// TwinCAT 3 PLC project BASF_RecipeCode_PLC
// ProgramVersion: 3.1.4022.4
// libraries:
//   Tc2_ModbusSrv, * (Beckhoff Automation GmbH)
//   Tc2_Standard, * (Beckhoff Automation GmbH)
//   Tc2_System, * (Beckhoff Automation GmbH)
//   Tc2_Utilities, * (Beckhoff Automation GmbH)
//   Tc3_Module, * (Beckhoff Automation GmbH)
// project tree:
//   AlarmUnit/ AlarmHandler.TcPOU, AlarmLogic.TcPOU, AlarmParametersProvider.TcPOU, DisableMaxAndMinAlarms.TcPOU
//   AlarmUnit/Structures/ AlarmParameters.TcDUT
//   DefaultValueCalculator/ GetDefaultValue.TcPOU
//   DUTs/ EachRecipeStep.TcDUT
//   GVL%27S/ Coupler.TcGVL (not stored), R1.TcGVL (not stored)
//   Helpers/ FB_Scaling.TcPOU, ScaledValueCalculator.TcPOU, LampStatusDecider.TcPOU, PossibilittyLogic.TcPOU, RemainingTimeCalculator.TcPOU, ShutDown.TcPOU
//   HuberHandlers/ HC_HUBER_1.TcPOU
//   JumoHelpers/ DataParser.TcPOU, ParameterParsingValue.TcPOU, StringSwapperForJumoRecorder.TcPOU
//   / Maintask.TcTTO, R1_task.TcTTO
//   POUs/ MAIN.TcPOU, PushToStartLogic.TcPOU
//   ReactorManager/AnalogScaling/ FB_AnalogScaling.TcPOU, I_AnalogScaling.TcIO
//   ReactorManager/ FB_Reactor.TcPOU
//   ReactorManager/HeatingCoolingMachineControl/ I_HeatCoolControl.TcIO
//   ReactorManager/Helpers/ Simulator.TcPOU
//   ReactorManager/MotorControl/ FB_MotorControl.TcPOU, I_MotorControl.TcIO
//   ReactorManager/MotorControl/MotorControlSupportModules/ FB_VfdIOControl.TcPOU
//   ReactorManager/RampLogic/ StirrerRampLogic.TcPOU
//   RecipeModules/ RecipeModule_R1.TcPOU, RecipeModule_R2.TcPOU, RecipeModule_R3.TcPOU, RecipeModule_R4.TcPOU, RecipeModule_R5.TcPOU, RecipeModule_R6.TcPOU

CONFIGURATION BASF_RecipeCode_PLC
    RESOURCE PLC ON TwinCAT3
        TASK Maintask(INTERVAL := T#25000us, PRIORITY := 2);
        TASK R1_task(INTERVAL := T#2ms, PRIORITY := 18);
        PROGRAM MAIN WITH Maintask : MAIN;
    END_RESOURCE
END_CONFIGURATION

// ---- AlarmUnit/Structures/AlarmParameters.TcDUT
TYPE AlarmParameters :
STRUCT
	CurrentParameterValue : REAL;
	MaxParameterLimit : REAL;
	MinParameterLimit : REAL;
	MaxLimitAlarm : BOOL;
	MinLimitAlarm : BOOL;
END_STRUCT
END_TYPE

// ---- DUTs/EachRecipeStep.TcDUT
TYPE EachRecipeStep :
STRUCT

   ///Tags for start block
     HeatCoolModeSelection:BOOL:=0; /// 0-is jacket mode/ 1-is process mode
	 HeatCoolDeltaTemp:DINT:=0; 
	 Started:BOOL:=0;
	 StartedTime:STRING:='';
	 Ended:BOOL:=0;
	 EndedTime:STRING:='';

	///Tags for HeatCoolBlock
	HeatCoolEnabled:BOOL:=0;
	HeatCoolStarted:BOOL:=0;
	HeatCoolStartedTime:STRING:='';
	HeatCoolEnded:BOOL:=0;
	HeatCoolEndedTime:STRING:='';
	HeatCoolSetPointExpression:DINT:=0;
	HeatCoolDuration:DINT:=0;
	HeatCoolOperatingMode:BOOL:=0;
	
	///Tags for StirrerBlock
	StirrerEnabled:BOOL:=0;
	StirrerStarted:BOOL:=0;
	StirrerStartedTime:STRING:='';
	StirrerEnded:BOOL:=0;
	StirrerEndedTime:STRING:='';
	StirrerSetPointExpression:DINT:=0;

	///Tags for DoseBlock	
	DosingEnabled:BOOL:=0;
	DosingStarted:BOOL:=0;
	DosingStartedTime:STRING:='';
	DosingEnded:BOOL:=0;
	DosingEndedTime:STRING:='';
    DosingMaxAmount:REAL:=0;
	DosingStopTemp:DINT:=0;
	DosingResumeTemp:DINT:=0;
	DosingRateSetpointExpression:REAL:=0;
	DosingMinRate:DINT:=0;
	DosingMaxRate:DINT:=0;
	DosingSettlingTime:DINT:=0;
	DosingMinPh:DINT:=0;
	DosingMaxPh:DINT:=0;
	DosingOperatingMode:BOOL:=0;
	
	////Tags for Wait tags
	WaitEnabled:BOOL:=0;
	WaitStarted:BOOL:=0;
	WaitStartedTime:STRING:='';
	WaitEndedTime:STRING:='';
	WaitEnded:BOOL:=0;
	WaitDuration:DINT:=0;
	WaitRemainingSeconds : INT;
	WaitRemainingMinutes : INT;
	WaitRemainingTime : STRING;
	
	//Tags for Centrifuge Block
	CentrifugeEnabled : BOOL;
	CentrifugeStarted : BOOL;
	CentrifugeEnded : BOOL;
	CentrifugeSpeedSetPoint : DINT;
	CentrifugeWaitTime : DINT;
	
	//Tags for Valves Block
	ValvesEnabled : BOOL;
	ValvesStarted : BOOL;
	ValvesEnded : BOOL;
	ValveAStatus : BOOL;
	ValveBStatus : BOOL;
	ValveCStatus : BOOL;
	
	//Tags for AOOD Pump Block
	AOODPumpEnabled : BOOL;
	AOODPumpStarted : BOOL;
	AOODPumpEnded : BOOL;
	Pump1Status : BOOL;
	Pump2Status : BOOL;

END_STRUCT
END_TYPE

// ---- ReactorManager/AnalogScaling/I_AnalogScaling.TcIO
INTERFACE I_AnalogScaling

METHOD ActualSpeed : REAL
VAR_INPUT
	nRawSensorValue		: REAL;
	nLowerScaleValue	: REAL;
	nHigherScaleValue	: REAL;
	nOutputLowerLimit	: REAL;
	nOutPutHigherLimit	: REAL;
END_VAR
END_METHOD

METHOD LoadCell : real
VAR_INPUT
	nRawSensorValue		: REAL;
	nLowerScaleValue	: REAL;
	nHigherScaleValue	: REAL;
	nOutputLowerLimit	: REAL;
	nOutPutHigherLimit	: REAL;
END_VAR
END_METHOD

METHOD pH : real
VAR_INPUT
	nRawSensorValue		: REAL;
	nLowerScaleValue	: REAL;
	nHigherScaleValue	: REAL;
	nOutputLowerLimit	: REAL;
	nOutPutHigherLimit	: REAL;
END_VAR
END_METHOD

METHOD Pressure : REAL
VAR_INPUT
	nRawSensorValue		: REAL;
	nLowerScaleValue	: REAL;
	nHigherScaleValue	: REAL;
	nOutputLowerLimit	: REAL;
	nOutPutHigherLimit	: REAL;
END_VAR
END_METHOD

METHOD Temperature : REAL
VAR_INPUT
	nRawSensorValue		: REAL;
	nLowerScaleValue	: REAL;
	nHigherScaleValue	: REAL;
	nOutputLowerLimit	: REAL;
	nOutPutHigherLimit	: REAL;
END_VAR
END_METHOD

END_INTERFACE

// ---- ReactorManager/HeatingCoolingMachineControl/I_HeatCoolControl.TcIO
INTERFACE I_HeatCoolControl

METHOD SetTemperature
VAR_INPUT
	nSetTemperature	: UINT;
END_VAR
END_METHOD

END_INTERFACE

// ---- ReactorManager/MotorControl/I_MotorControl.TcIO
INTERFACE I_MotorControl

METHOD GetActualSpeed : INT
END_METHOD

PROPERTY RemoteLocalStatus : bool
GET
END_GET
END_PROPERTY

METHOD SetSpeed : BOOL
VAR_INPUT
	nSetSpeed: INT;
END_VAR
END_METHOD

METHOD StartMotor : BOOL
VAR_INPUT
	bStart: BOOL;
END_VAR
END_METHOD

METHOD StopMotor : BOOL
VAR_INPUT
	bStop: BOOL;
END_VAR
END_METHOD

END_INTERFACE

// ---- POUs/MAIN.TcPOU
PROGRAM MAIN
VAR	 
	couplerConnectionStatus			: BOOL := TRUE;
	NullRecipeStepArray 			: ARRAY[0..100] OF EachRecipeStep;
	
	fglocal							: FB_LocalSystemTime;
	System_Time						: TIMESTRUCT;
	currentHour						: STRING;
	currentMinute					: STRING;
	concatenatedHourMinuteString	: STRING;
	scaledValueCalculator			: ScaledValueCalculator;
	ClearRecipeTrig_R1				: R_Trig;	
	
	fbAnalogScaling					: FB_AnalogScaling;
	ipAnalogScaling					: I_AnalogScaling	:= fbAnalogScaling;
	
	fbMotorControl					: FB_MotorControl;
	ipMotorControl					: I_MotorControl := fbMotorControl ;
	
	fbReactor						: FB_Reactor(ipAnalogScaling := ipAnalogScaling,ipMotorControl:= ipMotorControl);
END_VAR

VAR_INPUT
	ReactorEmergencyStatus AT %I* 	: ARRAY[1..6] OF BOOL;
END_VAR



// CALL THE REACTOR INSTANCE
fbReactor();



//Update Coupler Connection Status
IF	Coupler.CouplerConnectionState = 8 THEN
	Coupler.couplerConnectionStatus := TRUE;
ELSE
	Coupler.couplerConnectionStatus := FALSE; 
END_IF

//Code For Reading Current System Date and Time
fglocal(
	sNetID:='',
	bEnable:=TRUE,
	dwCycle:=5,
	dwOpt:=1,
	tTimeOut:=DEFAULT_ADS_TIMEOUT,
	bValid=> ,
	systemTime=>System_Time ,
	tzID=> );
	
//update current hour and minute strings	
currentHour := WORD_TO_STRING(fglocal.systemTime.wHour);
currentMinute := WORD_TO_STRING(fglocal.systemTime.wMinute);
concatenatedHourMinuteString := CONCAT(STR1:=currentHour, STR2:= ':');
concatenatedHourMinuteString := CONCAT(STR1:=concatenatedHourMinuteString, STR2:= currentMinute);

(* Update Used Now Status of Reactors and Other Equipment *)
IF R1.HeatCoolStatusFeedback OR R1.StirrerStatusFeedback THEN
	R1.UsedNow := TRUE;
ELSE	
	R1.UsedNow := FALSE;
END_IF

///CALL RECIPE MODULE-R1
IF R1.RecipeStatus THEN
	RecipeModule_R1();
END_IF
  
////End condition to wipe of the data in structure
	ClearRecipeTrig_R1(clk:=R1.ClearRecipe,q=>);
 IF ClearRecipeTrig_R1.Q  THEN
	R1.RecipeStatus:=FALSE;
	R1.RecipeStep := NullRecipeStepArray;
	R1.ClearRecipe:=FALSE;
	R1.RecipeEnded:=FALSE;
	R1.R1STEPS:=0;
	RecipeModule_R1.DosingTotalizerVolume:=0;
END_IF
   
//Stirre ramp
StirrerRampLogic();

END_PROGRAM

// ---- Helpers/ScaledValueCalculator.TcPOU
FUNCTION_BLOCK ScaledValueCalculator
VAR_INPUT
	nRawInputValue			: INT;
	nInputLowerLimit		: REAL;
	nInputHigherLimit		: REAL;
	nOutputLowerLimit		: REAL;
	nOutputHigherLimit		: REAL;
END_VAR
VAR_OUTPUT
		nScaledValueF		: REAL;
	    nScaledValueD		: INT;
END_VAR
VAR
	 nGain		: REAL;
END_VAR

// Scaling Calculations //

	IF	nRawInputValue	<	0	THEN
		nRawInputValue	:=	0;
	END_IF


	IF	 ((nInputHigherLimit - nInputLowerLimit)	<= 0)	OR
		 ((nOutputHigherLimit  - nOutputLowerLimit)	<= 0)	THEN
		nGain	:=	0;
	ELSE
		nGain:=(((nRawInputValue - nInputLowerLimit) / (nInputHigherLimit - nInputLowerLimit)) * (nOutputHigherLimit  - nOutputLowerLimit)) + nOutputLowerLimit;
	END_IF


		nScaledValueF	:=	nGain;
		nScaledValueD	:=	REAL_TO_INT(nGain);

END_FUNCTION_BLOCK

// ---- ReactorManager/AnalogScaling/FB_AnalogScaling.TcPOU
FUNCTION_BLOCK FB_AnalogScaling IMPLEMENTS I_AnalogScaling
VAR_INPUT
END_VAR
VAR_OUTPUT
END_VAR
VAR
		fbScaling		: FB_Scaling;
END_VAR

;

METHOD ActualSpeed : REAL
VAR_INPUT
	nRawSensorValue		: REAL;
	nLowerScaleValue	: REAL;
	nHigherScaleValue	: REAL;
	nOutputLowerLimit	: REAL;
	nOutPutHigherLimit	: REAL;
END_VAR
THIS^.fbScaling(
	nRawInputValue		:= nRawSensorValue, 
	nInputLowerLimit	:= nLowerScaleValue , 
	nInputHigherLimit	:= nHigherScaleValue, 
	nOutputLowerLimit	:= nOutputLowerLimit, 
	nOutputHigherLimit	:= nOutPutHigherLimit , 
	nScaledValueF		=> ActualSpeed, 
	nScaledValueD		=> );
END_METHOD

METHOD LoadCell : REAL
VAR_INPUT
	nRawSensorValue		: REAL;
	nLowerScaleValue	: REAL;
	nHigherScaleValue	: REAL;
	nOutputLowerLimit	: REAL;
	nOutPutHigherLimit	: REAL;
END_VAR
THIS^.fbScaling(
	nRawInputValue		:= nRawSensorValue, 
	nInputLowerLimit	:= nLowerScaleValue , 
	nInputHigherLimit	:= nHigherScaleValue, 
	nOutputLowerLimit	:= nOutputLowerLimit, 
	nOutputHigherLimit	:= nOutPutHigherLimit , 
	nScaledValueF		=> LoadCell, 
	nScaledValueD		=> );
END_METHOD

METHOD pH : REAL
VAR_INPUT
	nRawSensorValue		: REAL;
	nLowerScaleValue	: REAL;
	nHigherScaleValue	: REAL;
	nOutputLowerLimit	: REAL;
	nOutPutHigherLimit	: REAL;
END_VAR
THIS^.fbScaling(
	nRawInputValue		:= nRawSensorValue, 
	nInputLowerLimit	:= nLowerScaleValue , 
	nInputHigherLimit	:= nHigherScaleValue, 
	nOutputLowerLimit	:= nOutputLowerLimit, 
	nOutputHigherLimit	:= nOutPutHigherLimit , 
	nScaledValueF		=> pH, 
	nScaledValueD		=> );
END_METHOD

METHOD Pressure : REAL
VAR_INPUT
	nRawSensorValue		: REAL;
	nLowerScaleValue	: REAL;
	nHigherScaleValue	: REAL;
	nOutputLowerLimit	: REAL;
	nOutPutHigherLimit	: REAL;
END_VAR
THIS^.fbScaling(
	nRawInputValue		:= nRawSensorValue, 
	nInputLowerLimit	:= nLowerScaleValue , 
	nInputHigherLimit	:= nHigherScaleValue, 
	nOutputLowerLimit	:= nOutputLowerLimit, 
	nOutputHigherLimit	:= nOutPutHigherLimit , 
	nScaledValueF		=> Pressure, 
	nScaledValueD		=> );
END_METHOD

METHOD Temperature : REAL
VAR_INPUT
	nRawSensorValue		: REAL;
	nLowerScaleValue	: REAL;
	nHigherScaleValue	: REAL;
	nOutputLowerLimit	: REAL;
	nOutPutHigherLimit	: REAL;
END_VAR
THIS^.fbScaling(
	nRawInputValue		:= nRawSensorValue, 
	nInputLowerLimit	:= nLowerScaleValue , 
	nInputHigherLimit	:= nHigherScaleValue, 
	nOutputLowerLimit	:= nOutputLowerLimit, 
	nOutputHigherLimit	:= nOutPutHigherLimit , 
	nScaledValueF		=> Temperature, 
	nScaledValueD		=> );
END_METHOD

END_FUNCTION_BLOCK

// ---- Helpers/FB_Scaling.TcPOU
FUNCTION_BLOCK FB_Scaling
VAR_INPUT
	nRawInputValue: REAL;
	nInputLowerLimit: REAL;
	nInputHigherLimit: REAL;
	nOutputLowerLimit: REAL;
	nOutputHigherLimit: REAL;
END_VAR
VAR_OUTPUT
	nScaledValueF: REAL;
	nScaledValueD: INT;
END_VAR
VAR
	nGain: REAL;
END_VAR

// Scaling Calculations //

	IF	nRawInputValue	<	0	THEN
		nRawInputValue	:=	0;
	END_IF


	IF	 ((nInputHigherLimit - nInputLowerLimit)	<= 0)	OR
		 ((nOutputHigherLimit  - nOutputLowerLimit)	<= 0)	THEN
		nGain	:=	0;
	ELSE
		nGain:=(((nRawInputValue - nInputLowerLimit) / (nInputHigherLimit - nInputLowerLimit)) * (nOutputHigherLimit  - nOutputLowerLimit)) + nOutputLowerLimit;
	END_IF


		nScaledValueF	:=	nGain;
		nScaledValueD	:=	REAL_TO_INT(nGain);

END_FUNCTION_BLOCK

// ---- ReactorManager/MotorControl/FB_MotorControl.TcPOU
FUNCTION_BLOCK FB_MotorControl IMPLEMENTS I_MotorControl
VAR
	fbVfdIOControl: FB_VFDIOControl;
END_VAR

METHOD GetActualSpeed : INT
GetActualSpeed := fbVfdIOControl.nActualSpeed;
END_METHOD

PROPERTY RemoteLocalStatus : BOOL
GET
RemoteLocalStatus := fbVfdIOControl.bRemoteLocalStatus;
END_GET
END_PROPERTY

METHOD SetSpeed : BOOL
VAR_input
	nSetSpeed	: INT;
END_VAR
fbVfdIOControl.nSetSpeed := nSetSpeed;
END_METHOD

METHOD StartMotor : BOOL
VAR_INPUT
	bStart: BOOL;
END_VAR
fbVfdIOControl.bStartMotor := bStart;
END_METHOD

METHOD StopMotor : BOOL
VAR_INPUT
	bStop: BOOL;
END_VAR
fbVfdIOControl.bStopMotor := bStop;
END_METHOD

END_FUNCTION_BLOCK

// ---- ReactorManager/MotorControl/MotorControlSupportModules/FB_VfdIOControl.TcPOU
FUNCTION_BLOCK FB_VfdIOControl
VAR_INPUT
	bStartMotor			AT %Q*: BOOL;
	bStopMotor			AT %Q*: BOOL;
	nSetSpeed 			AT %Q*: INT;
	nActualSpeed		AT %I*: INT;
	bRemoteLocalStatus  AT %I* : BOOL;
END_VAR
VAR_OUTPUT
END_VAR
VAR

END_VAR

END_FUNCTION_BLOCK

// ---- ReactorManager/FB_Reactor.TcPOU
FUNCTION_BLOCK FB_Reactor
VAR_INPUT
	
END_VAR
VAR_OUTPUT
END_VAR
VAR
	simulator : Simulator;
	random_value : REAL;
	timeCounter : INT;
	updateAllParameters : BOOL;
	simulationMode : BOOL;
	
	ipMotorControl		: I_MotorControl;
	ipAnalogScaling		: I_AnalogScaling;
	nMassTemp AT %I*	: INT;
	nVentTemp AT %I*	: INT;
	nVapourTemp	AT %I*	: INT;
	nPressure AT %I*	: INT;
	nReactorpH AT %I*	: INT;
	nScrubberpH AT %I*	: INT;
	nLoadcell AT %I*	: INT;
	nStirrerSpeed AT %I*: INT;
	nLocalTemp			: REAL;
	nLocalTemp1			: REAL;
	nLocalTemp2			: REAL;
	nLocalTemp3 		: REAL;
	nLocalTemp4 		: REAL;
	nLocalTemp5 		: REAL;
	nLocalTemp6 		: REAL;
	nLocalTemp7 		: REAL;	
	nSpeedSetpoint 		: INT;
	nLocalSpeed			: REAL;
	fbScaling			: FB_Scaling;
END_VAR

IF simulationMode THEN
	IF updateAllParameters THEN
		random_value := 0;
		//Update parameters for R1 using Simulator logic
		random_value := 0;
		simulator(CurrentValue := R1.JacketOutletTemperature, TargetValue := DINT_TO_REAL(R1.HeatCoolSetPoint), SimulatedValue => random_value);
		R1.JacketOutletTemperature := REAL_TO_INT(random_value);
		
		simulator(CurrentValue := R1.ReactorMassTemperature, TargetValue := R1.JacketOutletTemperature, SimulatedValue => random_value);
		R1.ReactorMassTemperature := random_value;
		
		random_value := 0;
		simulator(CurrentValue := R1.StirrerCurrentSpeed, TargetValue := DINT_TO_REAL(R1.StirrerSetPoint), SimulatedValue => random_value);
		R1.StirrerCurrentSpeed := REAL_TO_INT(random_value);
		
		//Reset timeCounter
		updateAllParameters := FALSE;
		timeCounter := 0;
	ELSE
		timeCounter := timeCounter + 1;
		IF timeCounter >= 5 THEN
			updateAllParameters := TRUE;
		END_IF
	END_IF
ELSE
	//To Start Motor or Stop Motor
	(*Motor can be controlled from SCADA only if the Remote button is switched on from panel*)
	IF ipMotorControl.RemoteLocalStatus THEN //To check the panel remote status button
		IF R1.StirrerStatus THEN	
			//TO set the speed of the motor
			nLocalSpeed := R1.StirrerSetPoint*70.45;
			nSpeedSetpoint := TO_INT(nLocalSpeed)+6553;
			ipMotorControl.SetSpeed(nSpeedSetpoint);
		ELSE	
			ipMotorControl.SetSpeed(0);
		END_IF
	ELSE
		R1.StirrerStatus := FALSE;
	END_IF
	//========================================================================================================================================================================================================	
	//To call the Huber instance
	HC_HUBER_1();
	
	//Mass Temperature
	nLocalTemp	:= ipAnalogScaling.Temperature(nMassTemp,0,32767,-90,200);
	
	//Vent temp
	nLocalTemp1	:= ipAnalogScaling.Temperature(nVentTemp,0,32767,0,200);
	
	//Vapour temp
	nLocalTemp2	:= ipAnalogScaling.Temperature(nVapourTemp,0,32767,0,200);
	
	//Reactor pressure
	nLocalTemp3	:= ipAnalogScaling.Pressure(nPressure,0,32767,-1,1.5);
	
	//Reactor pH
	nLocalTemp4	:= ipAnalogScaling.pH(nReactorpH,0,32767,0,14);
	
	//Scrubber pH
	nLocalTemp5	:= ipAnalogScaling.pH(nScrubberpH,0,32767,0,14);
	
	//Load cell
	nLocalTemp6	:= ipAnalogScaling.LoadCell(nLoadcell,0,32767,0,150);
	
	//Stirrer actual speed
	nLocalTemp7	:= ipAnalogScaling.ActualSpeed(nLoadcell,0,32767,0,200);
	
		
	R1.ReactorMassTemperature	:= nLocalTemp ;
	R1.VentTemperature			:= nLocalTemp1 ;
	R1.VapourTemperature		:= nLocalTemp2 ;
	R1.Pressure					:= nLocalTemp3 ;
	R1.PHvalue					:= nLocalTemp4 ;
	R1.StirrerCurrentSpeed		:= TO_INT(nLocalTemp7);
	R1.ScrubberpH		:= nLocalTemp5;
	R1.ReactorMass				:= nLocalTemp6;
END_IF

METHOD FB_init : BOOL
VAR_INPUT
	bInitRetains	: BOOL; // if TRUE, the retain variables are initialized (warm start / cold start)
	bInCopyCode		: BOOL;  // if TRUE, the instance afterwards gets moved into the copy code (online change)
	ipMotorControl	: I_MotorControl;
	ipAnalogScaling	: I_AnalogScaling;
END_VAR
IF ipMotorControl <> 0 THEN
	THIS^.ipMotorControl := ipMotorControl;
END_IF

IF ipAnalogScaling <> 0 THEN
	THIS^.ipAnalogScaling := ipAnalogScaling;
END_IF
END_METHOD

END_FUNCTION_BLOCK

// ---- ReactorManager/Helpers/Simulator.TcPOU
FUNCTION_BLOCK Simulator
VAR_INPUT
	CurrentValue : REAL;
	TargetValue : REAL;
END_VAR
VAR_OUTPUT
	SimulatedValue : REAL;
END_VAR
VAR
	random_value : LREAL;
	fb_ran : DRAND;
END_VAR

fb_ran(Seed := 0, Num => random_value);
IF CurrentValue <= TargetValue THEN
	CurrentValue := CurrentValue + LREAL_TO_REAL(STRING_TO_LREAL(LREAL_TO_FMTSTR(random_value, 2, TRUE)));
ELSE
	CurrentValue := CurrentValue - LREAL_TO_REAL(STRING_TO_LREAL(LREAL_TO_FMTSTR(random_value, 2, TRUE)));
END_IF
SimulatedValue := STRING_TO_LREAL(LREAL_TO_FMTSTR(CurrentValue, 2, TRUE)); //Rounding again here to clear any errors above

END_FUNCTION_BLOCK

// ---- HuberHandlers/HC_HUBER_1.TcPOU
PROGRAM HC_HUBER_1
VAR	
	FcHC_2_Write_1	: FB_MBWriteSingleReg;
	FcHC_2_Write_2	: FB_MBWriteSingleReg;
	FcHC_2_Write_3	: FB_MBWriteSingleReg;
	FcHC_2_Write_4	: FB_MBWriteSingleReg;
	FcHC_2_Write_5	: FB_MBWriteSingleReg;
	FcHC_2_Write_6	: FB_MBWriteSingleReg;

	HCComp_2		: WORD;
	HCSelect_2		: WORD;
	HcCirc			: WORD;
	
	HCTempSetpoint_2		: WORD;
	HCReadParameters_2		: ARRAY[0..10] OF INT;

	HuberReadRegs_2			: FB_MBReadRegs;
	HuberReadTimer_2		: TON;
	HuberReadTimer_22		: TON;
	HuberWriteTimer_2		: TON;
	HuberWriteTimer_22		: TON;
END_VAR

//   HUBER_UNISTAT 510_2
//   HC
//   FUNCTION : DATA AQUISITION AND CONTROL
//   
//   COMMUNICATION WITH UNISTAT OVER MODBUS TCP
//   IP : 192.168.0.18


IF R1.HeatCoolStatus THEN 
	HCComp_2:=1;
	HcCirc:=1;
	ELSE
	HCComp_2:=0;
	HcCirc:=0;
END_IF

HCTempSetpoint_2:=DINT_TO_WORD(R1.HeatCoolSetPoint*100);

R1.HeatCoolStatusFeedback:=HCReadParameters_2[10].0;

R1.JacketOutletTemperature:=(INT_TO_REAL(HCReadParameters_2[1])/100);

///Select jacket/process 
IF R1.HeatCoolTemperatureControlType THEN
   HCSelect_2:=1;
   ELSE
   HCSelect_2:=0;	   
   END_IF





HuberReadTimer_2(IN:=NOT HuberReadTimer_22.Q , PT:=T#50MS, Q=> , ET=> );

HuberReadTimer_22(IN:=HuberReadTimer_2.Q , PT:=T#50MS , Q=> , ET=> );



///To read data  from the huber
HuberReadRegs_2(
	sIPAddr:='192.168.0.1' , 
	nTCPPort:=502 , 
	nUnitID:=1 , 
	nQuantity:=11 , 
	nMBAddr:=0 , 
	cbLength:=SIZEOF(HCReadParameters_2) , 
	pDestAddr:=ADR(HCReadParameters_2) , 
	bExecute:=HuberReadTimer_2.Q , 
	tTimeout:=T#5S , 
	bBusy=> , 
	bError=> , 
	nErrId=> , 
	cbRead=> );

HuberWriteTimer_2(IN:=NOT HuberWriteTimer_22.Q  , PT:=T#100MS , Q=> , ET=> );

HuberWriteTimer_22(IN:=HuberWriteTimer_2.Q , PT:=T#100MS, Q=> , ET=> );	
	
	
///To write temperature setpoint to the huber
FcHC_2_Write_1(
	sIPAddr:='192.168.0.1' , 
	nTCPPort:=502 , 
	nUnitID:=1 , 
	nMBAddr:=0 , 
	nValue:=HCTempSetpoint_2 , 
	bExecute:=HuberWriteTimer_2.Q , 
	tTimeout:=T#5S , 
	bBusy=> , 
	bError=> , 
	nErrId=> );	
	
/// jacket/ process selction	
	FcHC_2_Write_2(
	sIPAddr:='192.168.0.1' , 
	nTCPPort:=502 , 
	nUnitID:=1 , 
	nMBAddr:=19 , 
	nValue:=HCSelect_2 , 
	bExecute:=HuberWriteTimer_2.Q , 
	tTimeout:=T#5S , 
	bBusy=> , 
	bError=> , 
	nErrId=> );	
	
		
////To Switch on the machine	
	FcHC_2_Write_4(
	sIPAddr:='192.168.0.1' , 
	nTCPPort:=502 , 
	nUnitID:=1 , 
	nMBAddr:=20 , 
	nValue:=HCComp_2 , 
	bExecute:=HuberWriteTimer_2.Q , 
	tTimeout:=T#5S , 
	bBusy=> , 
	bError=> , 
	nErrId=> );	
	
	
///To switch on the circulation pump		
	FcHC_2_Write_5(
	sIPAddr:='192.168.0.1' , 
	nTCPPort:=502 , 
	nUnitID:=1 , 
	nMBAddr:=21 , 
	nValue:=HcCirc , 
	bExecute:=HuberWriteTimer_2.Q , 
	tTimeout:=T#5S , 
	bBusy=> , 
	bError=> , 
	nErrId=> );	
	
	
	IF 	FcHC_2_Write_5.bExecute OR 	FcHC_2_Write_4.bExecute OR 	FcHC_2_Write_3.bExecute OR 	FcHC_2_Write_2.bExecute OR 	FcHC_2_Write_1.bExecute OR HuberReadRegs_2.bExecute THEN 
///Error daignostics
	  IF HuberreadRegs_2.nErrId <> 0 OR FcHC_2_Write_1.nErrId <> 0 OR  FcHC_2_Write_2.nErrId <> 0 OR
	   FcHC_2_Write_3.nErrId <> 0 OR  FcHC_2_write_4.nErrId <> 0 THEN
	  R1.HeatCoolFailure:=TRUE;
	   ELSE
	  R1.HeatCoolFailure:=FALSE;
	 END_IF
	 END_IF

END_PROGRAM

// ---- RecipeModules/RecipeModule_R1.TcPOU
PROGRAM RecipeModule_R1
VAR
	shutDownFB:Shutdown;
	remainingTimeCalculator : RemainingTimeCalculator;
	
	DosingTick: INT;
	AbortTrig:R_Trig;
END_VAR
VAR_INPUT
	DosingTotalizerVolume: REAL;
END_VAR

IF R1.RecipeStep[0].Started AND R1.RecipeStep[0].StartedTime = '' THEN
	//Update StartedTime
	R1.RecipeStep[0].StartedTime := MAIN.concatenatedHourMinuteString;
END_IF

// Start Block and HC Mode Selection
IF R1.RecipeStep[R1.R1STEPS].Started THEN
  R1.R1STEPS:= R1.R1STEPS+1;
 // R1.AbortRecipe:=FALSE;
  R1.ClearRecipe:=FALSE;
  R1.RecipeEnded:=FALSE;
END_IF  
 
// Check Process or JACKET SELECTION
IF R1.RecipeStep[0].HeatCoolModeSelection THEN
	R1.HeatCoolTemperatureControlType:=TRUE;
	R1.TemperatureControl:=REAL_TO_DINT(R1.ReactorMassTemperature);
ELSE
	R1.HeatCoolTemperatureControlType:=FALSE;	
	R1.TemperatureControl:=REAL_TO_DINT(R1.JacketOutletTemperature);
END_IF

 IF R1.RecipeStep[R1.R1STEPS].HeatcoolEnabled THEN
	R1.HeatCoolSetPoint:=R1.RecipeStep[R1.R1STEPS].HeatCoolSetpointExpression;		
	R1.RecipeStep[R1.R1STEPS].HeatCoolStarted :=TRUE;
	IF R1.RecipeStep[R1.R1STEPS].HeatCoolStartedTime = '' THEN
		R1.RecipeStep[R1.R1STEPS].HeatCoolStartedTime := Main.concatenatedHourMinuteString;
	END_IF
	R1.HeatCoolStatus:=TRUE;
	
		///Check for condition in step  
	 IF ABS(R1.TemperatureControl-R1.RecipeStep[R1.R1STEPS].HeatCoolSetpointExpression )<0.5 THEN
		R1.RecipeStep[R1.R1STEPS].HeatcoolEnded :=TRUE;	
		IF R1.RecipeStep[R1.R1STEPS].HeatCoolEndedTime = '' THEN
			R1.RecipeStep[R1.R1STEPS].HeatCoolEndedTime := Main.concatenatedHourMinuteString;
		END_IF
	 END_IF     	
 END_IF
	
////Recipe block for stirrer
IF R1.RecipeStep[R1.R1STEPS].StirrerEnabled THEN
	R1.StirrerSetPoint:=R1.RecipeStep[R1.R1STEPS].StirrerSetPointExpression;
	R1.StirrerStatus:=TRUE;	
    R1.RecipeStep[R1.R1STEPS].StirrerStarted:=TRUE;
	IF R1.RecipeStep[R1.R1STEPS].StirrerStartedTime = '' THEN
		R1.RecipeStep[R1.R1STEPS].StirrerStartedTime := Main.concatenatedHourMinuteString;
	END_IF
	
	///Check the Actual speed to end the step
      IF ABS(R1.StirrerCurrentSpeed- R1.RecipeStep[R1.R1STEPS].StirrerSetPointExpression)<8 THEN
		R1.RecipeStep[R1.R1STEPS].StirrerEnded:=TRUE;
		IF R1.RecipeStep[R1.R1STEPS].StirrerEndedTime = '' THEN
			R1.RecipeStep[R1.R1STEPS].StirrerEndedTime := Main.concatenatedHourMinuteString;
		END_IF
	  END_IF
	//Check the rpm TO switch off the vfd
	  IF R1.RecipeStep[R1.R1STEPS].StirrerSetPointExpression=0 THEN
		R1.StirrerStatus:=FALSE;	
	  END_IF///
  END_IF 


(*////Wait Block*)
IF R1.RecipeStep[R1.R1STEPS].WaitEnabled AND NOT R1.RecipeStep[R1STEPS].WaitEnded THEN
    R1.RecipeStep[R1.R1STEPS].WaitStarted:=TRUE;
	IF R1.RecipeStep[R1.R1STEPS].WaitStartedTime = '' THEN
		R1.RecipeStep[R1.R1STEPS].WaitStartedTime := Main.concatenatedHourMinuteString;
	END_IF
	R1.WaitTick:=R1.WaitTick+1;
	IF R1.WaitTick=100  THEN
		//Update the Second Tick
		R1.WaitSecondTick:=R1.WaitSecondTick+1;
		R1.WaitTick:=0;
	END_IF
		
	IF  R1.WaitSecondTick=60  THEN
		//Update the Minute Tick
		R1.WaitMinuteTick:=R1.WaitMinuteTick+1;
		R1.WaitSecondTick:=0;
	END_IF	

	//Update the Remaining Time
	remainingTimeCalculator(elapsedSeconds:= R1.WaitSecondTick, elapsedMinutes:= R1.WaitMinuteTick, givenDuration:= DINT_TO_INT(R1.RecipeStep[R1.R1STEPS].WaitDuration), 
							leftOverSeconds=> R1.RecipeStep[R1.R1STEPS].WaitRemainingSeconds, leftOverMinutes=> R1.RecipeStep[R1.R1STEPS].WaitRemainingMinutes);
	R1.RecipeStep[R1.R1STEPS].WaitRemainingTime := INT_TO_STRING(R1.RecipeStep[R1.R1STEPS].WaitRemainingMinutes);
	R1.RecipeStep[R1.R1STEPS].WaitRemainingTime := CONCAT(STR1:= R1.RecipeStep[R1.R1STEPS].WaitRemainingTime, STR2:= ':');
	R1.RecipeStep[R1.R1STEPS].WaitRemainingTime := CONCAT(STR1:= R1.RecipeStep[R1.R1STEPS].WaitRemainingTime, STR2:= INT_TO_STRING(R1.RecipeStep[R1.R1STEPS].WaitRemainingSeconds));
	
	(*///To write ended time*)
	IF ABS(R1.WaitMinuteTick -R1.RecipeStep[R1.R1STEPS].WaitDuration)=0 THEN
		R1.RecipeStep[R1.R1STEPS].WaitEnded:=TRUE;
		IF R1.RecipeStep[R1.R1STEPS].WaitEndedTime = '' THEN
			R1.RecipeStep[R1.R1STEPS].WaitEndedTime := Main.concatenatedHourMinuteString;
		END_IF
		R1.WaitTick:=0;
		R1.WaitSecondTick:=0;
		R1.WaitMinuteTick:=0;
	END_IF
END_IF
	
IF R1.RecipeStep[R1STEPS].DosingEnabled AND NOT R1.RecipeStep[R1STEPS].DosingEnded THEN
	R1.RecipeStep[R1STEPS].DosingStarted := TRUE;
	IF R1.RecipeStep[R1.R1STEPS].DosingStartedTime = '' THEN
		R1.RecipeStep[R1.R1STEPS].DosingStartedTime := Main.concatenatedHourMinuteString;
	END_IF
	//Update Totalized Volume
		IF  R1.DosingPumpStatus_1 THEN
			DosingTick:=DosingTick+1;
		END_IF
		   
	  IF DosingTick=100 THEN
		  DosingTotalizerVolume:=DosingTotalizerVolume+(R1.RecipeStep[R1STEPS].DosingRateSetpointExpression/2.7 * 0.045);	  
	  END_IF
	  
	  IF DosingTick>100 THEN
		  DosingTick:=0;
	  END_IF
	  
	IF DosingTotalizerVolume < R1.RecipeStep[R1STEPS].DosingMaxAmount THEN
		IF R1.DosingPumpStatus_1 THEN
			IF R1.TemperatureControl < R1.RecipeStep[R1STEPS].DosingStopTemp THEN
				R1.DosingPumpStatus_1 := TRUE;
				R1.DosingPumpSetPoint_1 := R1.RecipeStep[R1STEPS].DosingRateSetpointExpression;
			ELSE
				R1.DosingPumpStatus_1 := FALSE;
				R1.DosingPumpSetPoint_1 := 0;
			END_IF
		ELSE
			IF DosingTotalizerVolume = 0 AND R1.TemperatureControl > R1.RecipeStep[R1STEPS].DosingResumeTemp AND R1.TemperatureControl < R1.RecipeStep[R1STEPS].DosingStopTemp THEN
				//Logic for starting Dosing Pump First Time in a Recipe Step
				R1.DosingPumpStatus_1 := TRUE;
				R1.DosingPumpSetPoint_1 := R1.RecipeStep[R1STEPS].DosingRateSetpointExpression;
			END_IF
			
			IF R1.TemperatureControl < R1.RecipeStep[R1STEPS].DosingResumeTemp THEN
				R1.DosingPumpStatus_1 := TRUE;
				R1.DosingPumpSetPoint_1 := R1.RecipeStep[R1STEPS].DosingRateSetpointExpression;
			END_IF
		END_IF
	ELSE
		R1.DosingPumpStatus_1 := FALSE;
		R1.DosingPumpSetPoint_1 := 0;
		R1.RecipeStep[R1STEPS].DosingEnded := TRUE;
		IF R1.RecipeStep[R1.R1STEPS].DosingEndedTime = '' THEN
			R1.RecipeStep[R1.R1STEPS].DosingEndedTime := Main.concatenatedHourMinuteString;
		END_IF
		DosingTick := 0;
		DosingTotalizerVolume:=0;
	END_IF
END_IF

IF R1.R1STEPS>0 THEN 

(*//Step control block To increment to next step*)
 R1.TotalEnabledValue:=BOOL_TO_INT(R1.RecipeStep[R1.R1STEPS].HeatcoolEnabled)+BOOL_TO_INT(R1.RecipeStep[R1.R1STEPS].StirrerEnabled)+BOOL_TO_INT(R1.RecipeStep[R1.R1STEPS].WaitEnabled)+BOOL_TO_INT( R1.RecipeStep[R1.R1STEPS].DosingEnabled);
 R1.TotalEndedValue:=BOOL_TO_INT(R1.RecipeStep[R1.R1STEPS].HeatCoolEnded)+BOOL_TO_INT(R1.RecipeStep[R1.R1STEPS].StirrerEnded)+BOOL_TO_INT(R1.RecipeStep[R1.R1STEPS].WaitEnded)+BOOL_TO_INT( R1.RecipeStep[R1.R1STEPS].DosingEnded);

    IF (R1.TotalEnabledValue - R1.TotalEndedValue)=0 THEN 
		R1.R1STEPS:=R1.R1STEPS+1;
    END_IF
END_IF
  
 (* ///To End the Recipe**)
 IF  R1.NumberOfRecipeSteps = R1.R1STEPS THEN
	 R1.StirrerStatus:=FALSE;
	 R1.StirrerSetPoint:=0;
	 R1.HeatCoolStatus:=FALSE;
	 R1.HeatCoolSetPoint:=0;	
     R1.StepCompleted:=FALSE;	 
	 R1.RecipeEnded:=TRUE;
	 R1.RecipeStatus:=FALSE;
 END_IF
  
(* //TO ABORT RECIPE*)
AbortTrig(CLK:=R1.AbortRecipe,Q=>);
IF AbortTrig.Q THEN
	shutDownFB(GvlIdentifier := 'R1');
	AbortTrig.CLK := FALSE;
END_IF

END_PROGRAM

// ---- Helpers/ShutDown.TcPOU
FUNCTION_BLOCK PUBLIC ShutDown
VAR_INPUT
	GvlIdentifier : STRING;
END_VAR
VAR_OUTPUT
END_VAR
VAR
END_VAR

IF GvlIdentifier = 'R1' THEN
	R1.RecipeStatus		:= FALSE;
	R1.HeatCoolStatus	:= FALSE;
	R1.StirrerStatus	:= FALSE;
	R1.AbortRecipe		:= FALSE;
END_IF;

END_FUNCTION_BLOCK

// ---- Helpers/RemainingTimeCalculator.TcPOU
FUNCTION_BLOCK PUBLIC RemainingTimeCalculator
VAR_INPUT
	elapsedSeconds : INT;
	elapsedMinutes : INT;
	givenDuration : INT; //Assume Duration in Minutes by default
END_VAR
VAR_OUTPUT
	leftOverSeconds : INT;
	leftOverMinutes : INT;
END_VAR
VAR
END_VAR

IF givenDuration <= elapsedMinutes THEN
	leftOverSeconds := 0;
	leftOverMinutes := 0;
ELSE
	leftOverMinutes := givenDuration - elapsedMinutes - 1;
	leftOverSeconds := 60 - elapsedSeconds;
END_IF

END_FUNCTION_BLOCK

// ---- ReactorManager/RampLogic/StirrerRampLogic.TcPOU
PROGRAM StirrerRampLogic

VAR
	i: INT;
	rTime : STRING;
	rMin : DINT;
	rSec : INT;
END_VAR


//// ramp for stirrer R1
IF R1.StirrerStartTimer=1 THEN
	

R1.StirrerTick:=R1.StirrerTick+1;

IF R1.StirrerTick=40  THEN
	R1.StirrerSecondTick:=R1.StirrerSecondTick+1;
	R1.StirrerTick:=0;
END_IF

IF R1.StirrerSecondTick=60  THEN
	R1.StirrerMinuteTick:=R1.StirrerMinuteTick+1;
	R1.StirrerSecondTick:=0;
END_IF

ELSE
	R1.StirrerTick:=0;
	R1.StirrerSecondTick:=0;
	R1.StirrerMinuteTick:=0;
END_IF
// START RAMP

IF R1.StirrerRampStatus THEN
	//initialize ramp parameters if first step
	IF R1.StirrerRampStep = -1 THEN
		R1.StirrerRampStep := R1.StirrerRampStep + 1;
		R1.StirrerRampStarted[R1.StirrerRampStep]:=TRUE;
		R1.StirrerRampStartedTime[R1.StirrerRampStep]:= Main.concatenatedHourMinuteString;
	END_IF
	
	R1.StirrerStatus := TRUE;
	// WRITE RAMP SP TO Stirrer SP	
	R1.StirrerSetPoint:=R1.StirrerRampSetpoint[R1.StirrerRampStep];
	// CHECK IF RPM REACHES SP
	IF ABS(R1.StirrerCurrentSpeed-R1.StirrerRampSetpoint[R1.StirrerRampStep])<5 THEN
		R1.StirrerSPCheck:=1;
		ELSE
		R1.StirrerSPCheck:=0;
	END_IF
	
	R1.StirrerSPCheck_R(CLK:=R1.StirrerSPCheck , Q=>R1.StirrerSPChecktrigger );
	// IF SP REACHED START TIMER
	IF R1.StirrerSPChecktrigger THEN
	R1.StirrerStartTimer:=1;
		
	END_IF
	// CHECK IF HOLD TIME ELAPSED. IF ELAPSED CHECK IF LAST STEP AND END ELSE INCREMENT STEP
	IF (R1.StirrerMinuteTick-R1.StirrerRampTime[R1.StirrerRampStep])=0 THEN
		  R1.StirrerRampEnded[R1.StirrerRampStep]:=1;
		  IF R1.StirrerRampEndedTime[R1.StirrerRampStep] = '' THEN
			 R1.StirrerRampEndedTime[R1.StirrerRampStep]:= Main.concatenatedHourMinuteString;
		  END_IF
		  R1.StirrerRampStep:=R1.StirrerRampStep+1;
		  IF R1.StirrerRampStep=R1.StirrerRampNumberOfSteps THEN
			  R1.StirrerRampStatus:=0;
			  R1.StirrerStartTimer:=0;  
			  ELSE
				R1.StirrerRampStarted[R1.StirrerRampStep]:=1;
				IF R1.StirrerRampStartedTime[R1.StirrerRampStep] = '' THEN
					R1.StirrerRampStartedTime[R1.StirrerRampStep]:= Main.concatenatedHourMinuteString;
				END_IF
				R1.StirrerMinuteTick:=0;
				R1.StirrerStartTimer:=0;  
		  END_IF
	END_IF
	
	//update the remaining time in current step
	rMin := R1.StirrerRampTime[R1.StirrerRampStep] - R1.StirrerMinuteTick - 1;
	IF rMin < 0 THEN
		rMin := 0;
	END_IF
	rSec := 60 - R1.StirrerSecondTick;
	IF rSec = 0 THEN
		rMin := rMin + 1;
	END_IF
	R1.StirrerRampRemainingTime := concat(DINT_TO_STRING(rMin), ':');
	R1.StirrerRampRemainingTime := concat(R1.StirrerRampRemainingTime, DINT_TO_STRING(rSec));
	
	// SKIP OPERATION . IF SKIP PRESSED THEN INCREMENT STEP AFTER CHECKING BOUNDARY CONDN
	R1.StirrerRampSkip(CLK:=R1.StirrerRampStepSkipStatus , Q=>R1.StirrerRampSkipTrigger );
	IF R1.StirrerRampSkipTrigger AND R1.StirrerRampStep<=(R1.StirrerRampNumberOfSteps - 1) THEN
		R1.StirrerRampStepSkipStatus := FALSE; //reset the bit set true by SCADA
		R1.StirrerRampEnded[R1.StirrerRampStep]:=1;
		R1.StirrerRampEndedTime[R1.StirrerRampStep]:= Main.concatenatedHourMinuteString;
		IF R1.StirrerRampStep < R1.StirrerRampNumberOfSteps THEN
			R1.StirrerRampStep:=R1.StirrerRampStep+1;
			R1.StirrerStartTimer:=0;
			R1.StirrerRampStarted[R1.StirrerRampStep]:=1;
			R1.StirrerRampStartedTime[R1.StirrerRampStep]:=Main.concatenatedHourMinuteString;
		ELSE
			// we are in the last step of Ramp. So turn the RampStatus off.
			R1.StirrerRampStatus := FALSE;
		END_IF
	END_IF
	
	// EDIT OPERATION
	R1.StirrerRampEdit(CLK:=R1.StirrerRampStepEditStatus , Q=>R1.StirrerRampEditTrigger );
	IF R1.StirrerRampEditTrigger THEN
		//reset the timer so the step will start again
		R1.StirrerStartTimer:=0;  
	END_IF
	
	R1.StirrerRampClear(clk:= R1.StirrerRampClearStatus, q=>R1.StirrerRampClearStatus);
	IF R1.StirrerRampClearTrigger THEN
		R1.StirrerRampClearStatus := FALSE; //reset the bit set true by SCADA
		R1.StirrerRampStep:=-1;
		R1.StirrerRampStartedTime[i]:='';
		R1.StirrerRampEndedTime[i]:='';
	END_IF
ELSE
	R1.StirrerRampStep:=-1;
	R1.StirrerRampRemainingTime := '';
	FOR i:= 0 TO 7 DO
		R1.StirrerRampStarted[i]:=FALSE;
		R1.StirrerRampEnded[i]:=FALSE;
	END_FOR
END_IF

END_PROGRAM

// ---- AlarmUnit/AlarmHandler.TcPOU
PROGRAM AlarmHandler
VAR
	alarmLogic : AlarmLogic;
	disableAlarms : DisableMaxAndMinAlarms;
END_VAR

IF R1.AlarmsEnabled AND R1.RunningBatchStatus THEN
	alarmLogic(GivenParameterArray := AlarmParametersProvider(CurrentParameterValue := R1.ReactorMassTemperature, MaxParameterLimit := R1.HCTempMaxLimit, MinParameterLimit := R1.HCTempMinLimit),
			   MaxLimitExceeded =>	R1.HCTempMaxLimitExceeded, MinLimitExceeded => R1.HCTempMinLimitExceeded);
		
    alarmLogic(GivenParameterArray := AlarmParametersProvider(CurrentParameterValue := R1.JacketOutletTemperature, MaxParameterLimit := R1.JacketTempMaxLimit, MinParameterLimit := R1.JacketTempMinLimit),
			   MaxLimitExceeded =>	R1.JacketTempMaxLimitExceeded, MinLimitExceeded => R1.jacketTempMinLimitExceeded);	   
ELSE
	(* Disable alarms *)
	disableAlarms(MaxAlarmStatus => R1.HCTempMaxLimitExceeded, MinAlarmStatus => R1.HCTempMinLimitExceeded);
	disableAlarms(MaxAlarmStatus => R1.JacketTempMaxLimitExceeded, MinAlarmStatus => R1.JacketTempMinLimitExceeded);
END_IF


///Reactor-2
IF R2.AlarmsEnabled AND R2.RunningBatchStatus THEN
	alarmLogic(GivenParameterArray := AlarmParametersProvider(CurrentParameterValue := R2.ReactorMassTemperature, MaxParameterLimit := R2.HCTempMaxLimit, MinParameterLimit := R2.HCTempMinLimit),
			   MaxLimitExceeded =>	R2.HCTempMaxLimitExceeded, MinLimitExceeded => R2.HCTempMinLimitExceeded);
			   
    alarmLogic(GivenParameterArray := AlarmParametersProvider(CurrentParameterValue := R2.JacketOutletTemperature, MaxParameterLimit := R2.JacketTempMaxLimit, MinParameterLimit := R2.JacketTempMinLimit),
			   MaxLimitExceeded =>	R2.JacketTempMaxLimitExceeded, MinLimitExceeded => R2.JacketTempMinLimitExceeded);			   
ELSE
	(* Disable alarms *)
	disableAlarms(MaxAlarmStatus => R2.HCTempMaxLimitExceeded, MinAlarmStatus => R2.HCTempMinLimitExceeded);
	disableAlarms(MaxAlarmStatus => R2.JacketTempMaxLimitExceeded, MinAlarmStatus => R2.JacketTempMinLimitExceeded);
END_IF



///Reactor-3
IF R3.AlarmsEnabled AND R3.RunningBatchStatus THEN
	alarmLogic(GivenParameterArray := AlarmParametersProvider(CurrentParameterValue := R3.ReactorMassTemperature, MaxParameterLimit := R3.HCTempMaxLimit, MinParameterLimit := R3.HCTempMinLimit),
			   MaxLimitExceeded =>	R3.HCTempMaxLimitExceeded, MinLimitExceeded => R3.HCTempMinLimitExceeded);
			   
    alarmLogic(GivenParameterArray := AlarmParametersProvider(CurrentParameterValue := R3.JacketOutletTemperature, MaxParameterLimit := R3.JacketTempMaxLimit, MinParameterLimit := R3.JacketTempMinLimit),
			   MaxLimitExceeded =>	R3.JacketTempMaxLimitExceeded, MinLimitExceeded => R3.JacketTempMinLimitExceeded);			   
ELSE
	(* Disable alarms *)
	disableAlarms(MaxAlarmStatus => R3.HCTempMaxLimitExceeded, MinAlarmStatus => R3.HCTempMinLimitExceeded);
	disableAlarms(MaxAlarmStatus => R3.JacketTempMaxLimitExceeded, MinAlarmStatus => R3.JacketTempMinLimitExceeded);
END_IF



///Reactor-4
IF R4.AlarmsEnabled AND R4.RunningBatchStatus THEN
	alarmLogic(GivenParameterArray := AlarmParametersProvider(CurrentParameterValue := R4.ReactorMassTemperature, MaxParameterLimit := R4.HCTempMaxLimit, MinParameterLimit := R4.HCTempMinLimit),
			   MaxLimitExceeded =>	R4.HCTempMaxLimitExceeded, MinLimitExceeded => R4.HCTempMinLimitExceeded);
			   
    alarmLogic(GivenParameterArray := AlarmParametersProvider(CurrentParameterValue := R4.JacketOutletTemperature, MaxParameterLimit := R4.JacketTempMaxLimit, MinParameterLimit := R4.JacketTempMinLimit),
			   MaxLimitExceeded =>	R4.JacketTempMaxLimitExceeded, MinLimitExceeded => R4.JacketTempMinLimitExceeded);			   
ELSE
	(* Disable alarms *)
	disableAlarms(MaxAlarmStatus => R4.HCTempMaxLimitExceeded, MinAlarmStatus => R4.HCTempMinLimitExceeded);
	disableAlarms(MaxAlarmStatus => R4.JacketTempMaxLimitExceeded, MinAlarmStatus => R4.JacketTempMinLimitExceeded);
END_IF




///Reactor-5
IF R5.AlarmsEnabled AND R5.RunningBatchStatus THEN
	alarmLogic(GivenParameterArray := AlarmParametersProvider(CurrentParameterValue := R5.ReactorMassTemperature, MaxParameterLimit := R5.HCTempMaxLimit, MinParameterLimit := R5.HCTempMinLimit),
			   MaxLimitExceeded =>	R5.HCTempMaxLimitExceeded, MinLimitExceeded => R5.HCTempMinLimitExceeded);
			   
    alarmLogic(GivenParameterArray := AlarmParametersProvider(CurrentParameterValue := R5.JacketOutletTemperature, MaxParameterLimit := R5.JacketTempMaxLimit, MinParameterLimit := R5.JacketTempMinLimit),
			   MaxLimitExceeded =>	R5.JacketTempMaxLimitExceeded, MinLimitExceeded => R5.JacketTempMinLimitExceeded);			   
ELSE
	(* Disable alarms *)
	disableAlarms(MaxAlarmStatus => R5.HCTempMaxLimitExceeded, MinAlarmStatus => R5.HCTempMinLimitExceeded);
	disableAlarms(MaxAlarmStatus => R5.JacketTempMaxLimitExceeded, MinAlarmStatus => R5.JacketTempMinLimitExceeded);
END_IF




///Reactor-6
IF R6.AlarmsEnabled AND R6.RunningBatchStatus THEN
	alarmLogic(GivenParameterArray := AlarmParametersProvider(CurrentParameterValue := R6.ReactorMassTemperature, MaxParameterLimit := R6.HCTempMaxLimit, MinParameterLimit := R6.HCTempMinLimit),
			   MaxLimitExceeded =>	R6.HCTempMaxLimitExceeded, MinLimitExceeded => R6.HCTempMinLimitExceeded);
			   
    alarmLogic(GivenParameterArray := AlarmParametersProvider(CurrentParameterValue := R6.JacketOutletTemperature, MaxParameterLimit := R6.JacketTempMaxLimit, MinParameterLimit := R6.JacketTempMinLimit),
			   MaxLimitExceeded =>	R6.JacketTempMaxLimitExceeded, MinLimitExceeded => R6.JacketTempMinLimitExceeded);			   
ELSE
	(* Disable alarms *)
	disableAlarms(MaxAlarmStatus => R6.HCTempMaxLimitExceeded, MinAlarmStatus => R6.HCTempMinLimitExceeded);
	disableAlarms(MaxAlarmStatus => R6.JacketTempMaxLimitExceeded, MinAlarmStatus => R6.JacketTempMinLimitExceeded);
END_IF

END_PROGRAM

// ---- AlarmUnit/AlarmLogic.TcPOU
FUNCTION_BLOCK PUBLIC AlarmLogic
VAR_INPUT
	GivenParameterArray : AlarmParameters;
END_VAR
VAR_OUTPUT
	MaxLimitExceeded : BOOL;
	MinLimitExceeded : BOOL;
END_VAR
VAR
END_VAR

(*
Check if Exceeded bit(Max or Min) was false initially then only write True to Exceeded bit
because overwriting True leads to unnecessary notifications from Plc to Application
*)
IF GivenParameterArray.CurrentParameterValue > GivenParameterArray.MaxParameterLimit AND NOT MaxLimitExceeded THEN
	MaxLimitExceeded := TRUE;
	MinLimitExceeded := FALSE;
ELSIF GivenParameterArray.CurrentParameterValue < GivenParameterArray.MinParameterLimit AND NOT MinLimitExceeded THEN
	MaxLimitExceeded := FALSE;
	MinLimitExceeded := TRUE;
ELSIF GivenParameterArray.CurrentParameterValue <= GivenParameterArray.MaxParameterLimit AND GivenParameterArray.CurrentParameterValue >= GivenParameterArray.MinParameterLimit THEN
	(* Disable the Exceeded bits if current parameter value lies between Max and Min Limits *)
	MaxLimitExceeded := FALSE;
	MinLimitExceeded := FALSE;
END_IF

END_FUNCTION_BLOCK

// ---- AlarmUnit/DisableMaxAndMinAlarms.TcPOU
FUNCTION_BLOCK PUBLIC DisableMaxAndMinAlarms
VAR_INPUT
END_VAR
VAR_OUTPUT
	(* As name suggest force write the Max and Min alarms false *)
	MaxAlarmStatus : BOOL := FALSE;
	MinAlarmStatus : BOOL := FALSE;
END_VAR
VAR
END_VAR

END_FUNCTION_BLOCK

// ---- AlarmUnit/AlarmParametersProvider.TcPOU
FUNCTION AlarmParametersProvider : AlarmParameters
VAR_INPUT
	CurrentParameterValue : REAL;
	MaxParameterLimit : REAL;
	MinParameterLimit : REAL;
END_VAR
VAR
	alarmParameters : AlarmParameters;
END_VAR

alarmParameters.CurrentParameterValue := CurrentParameterValue;
alarmParameters.MaxParameterLimit := MaxParameterLimit;
alarmParameters.MinParameterLimit := MinParameterLimit;

AlarmParametersProvider := alarmParameters;

END_FUNCTION

// ---- DefaultValueCalculator/GetDefaultValue.TcPOU
FUNCTION GetDefaultValue : string
VAR_INPUT
	DataType : STRING;
END_VAR
VAR
	defaultValue : STRING;
END_VAR

IF DataType = 'string' THEN
	defaultValue := '';
END_IF

GetDefaultValue := defaultValue;

END_FUNCTION

// ---- Helpers/LampStatusDecider.TcPOU
FUNCTION_BLOCK PUBLIC LampStatusDecider
VAR_INPUT
	GivenTimer : TON;
	GivenTimer_1: TON;
	Giventimer_2: TON;
	
	CurrentStatus : BOOL;
END_VAR
VAR_OUTPUT
	NewStatus : BOOL;
END_VAR
VAR
END_VAR



	GivenTimer_1(IN:= NOT Giventimer_2.Q,PT:=T#500MS,Q=> );
	
	GivenTimer_2(IN:=GivenTimer_1.Q,PT:=T#500ms,Q=>);
	
	IF GivenTimer_1.Q THEN
	   NewStatus:=TRUE;	
	   ELSE
	   NewStatus:=FALSE;	   
	   END_IF
	
	




//IF GivenTimer.Q THEN
	//NewStatus := NOT CurrentStatus;
//END_IF

END_FUNCTION_BLOCK

// ---- Helpers/PossibilittyLogic.TcPOU
FUNCTION_BLOCK PossibilittyLogic
VAR_INPUT
	TriggerInput:BOOL;
END_VAR
VAR_OUTPUT
	TriggerOutput:BOOL;
END_VAR
VAR
	Counter:INT;
	FalseCounter:int;
	TriggerON:R_TRIG;
	TriggerOFF:F_Trig;
END_VAR


///Increment the counter when the bit is high
TriggerON(CLK:=TriggerInput,q=>);
IF TriggerON.Q THEN
  TriggerOutput:=TRUE;
  FalseCounter:=0;
END_IF
///Decrement the counter when the bit is low
//Increment the countier if the input is continoussly low
IF TriggerInput=FALSE THEN
   FalseCounter:=FalseCounter+1;
   IF  FalseCounter>1000 THEN
	   falseCounter:=0;
   END_IF
END_IF

IF FalseCounter>700 THEN
   TriggerOutput:=FALSE;   
   END_IF

END_FUNCTION_BLOCK

// ---- JumoHelpers/DataParser.TcPOU
FUNCTION_BLOCK PUBLIC DataParser
VAR_INPUT
	GivenArray : ARRAY[0..5] OF REAL;
END_VAR
VAR_OUTPUT
	OutputArray : ARRAY[0..5] OF REAL;
END_VAR
VAR
	i : INT;
END_VAR

FOR i:= 0 TO 5 BY 1 DO
    OutputArray[i] := ParameterParsingValue(GivenArray[i]);
END_FOR;

END_FUNCTION_BLOCK

// ---- JumoHelpers/ParameterParsingValue.TcPOU
FUNCTION ParameterParsingValue : REAL
VAR_INPUT
	InputParameter:REAL;
END_VAR	
VAR
	ParsedStringValue:STRING;
	
END_VAR

//Rounding up the given parameter 
ParsedStringValue:=Lreal_to_fmtstr(InputParameter,1,TRUE);

//Converting  String to real

ParameterParsingValue:=STRING_TO_REAL(ParsedStringValue);

END_FUNCTION

// ---- JumoHelpers/StringSwapperForJumoRecorder.TcPOU
FUNCTION StringSwapperForJumoRecorder : STRING
VAR_INPUT
	GivenString : STRING;
END_VAR
VAR
	i : INT;
	tempString : STRING;
	finalSwappedString : STRING;
	lengthOfGivenString : INT := Len(GivenString);
	tempChar : STRING(255);
END_VAR

IF (lengthOfGivenString MOD 2) <> 0 THEN
	GivenString := concat(GivenString, ' ');
END_IF

FOR i:=1 TO Len(GivenString) BY 2 DO
    IF mid(GivenString, 1, i) = ' ' THEN
		tempString := replace(tempString, ' ', 1, i);
	ELSE
		tempString := replace(tempString, mid(GivenString, 1, i), 1, i);
	END_IF
	
	IF mid(GivenString, 1, i + 1) = ' ' THEN
		tempString := replace(tempString, ' ', 1, i + 1);
	ELSE
		tempString := replace(tempString, mid(GivenString, 1, i + 1), 1, i + 1);
	END_IF
	
	tempChar := mid(tempString, 1, i);
	tempString := replace(tempString, mid(tempString, 1, i + 1), 1, i);
	tempString := replace(tempString, tempChar, 1, i + 1);
	
	finalSwappedString := concat(finalSwappedString, mid(tempString, 1, i));
	finalSwappedString := concat(finalSwappedString, mid(tempString, 1, i + 1));
END_FOR;

StringSwapperForJumoRecorder := finalSwappedString;

END_FUNCTION

// ---- POUs/PushToStartLogic.TcPOU
FUNCTION_BLOCK PushToStartLogic
VAR_INPUT
	StartEquipment:BOOL;
END_VAR
VAR_OUTPUT
	RelayCommandToStart:BOOL;
	RelayCommandToStop:BOOL;
END_VAR
VAR
     StartTrig:R_Trig;
	 Stoptrig:F_Trig;
	
	 StartCounter:INT;
	 StopCounter:INT;	
END_VAR

///Logic for the push button

///Start logic 
StartTrig(CLK:=StartEquipment,q=>);

IF StartTrig.Q THEN
   RelayCommandToStart:=TRUE;
END_IF

IF RelayCommandToStart THEN
   StartCounter:=StartCounter+1;
IF StartCounter=50 THEN
   RelayCommandToSTart:=FALSE;	
   StartCounter:=0;
END_IF
END_IF
   
 ///Stop logic
 StopTrig(CLK:=StartEquipmenT,Q=>);
 IF StopTrig.Q THEN
	RelayCommandToStop:=TRUE;
 END_IF
 
 IF RelayCommandToStop THEN
	StopCounter:=StopCounter+1;
    IF StopCounter=50 THEN
	   RelayCommandToStop:=FALSE;
	   StopCounter:=0;
    END_IF
 END_IF

END_FUNCTION_BLOCK

// ---- RecipeModules/RecipeModule_R2.TcPOU
PROGRAM RecipeModule_R2
VAR
	shutDownFB:Shutdown;
	remainingTimeCalculator : RemainingTimeCalculator;
	
	DosingTick: INT;
	AbortTrig:R_Trig;
END_VAR
VAR_INPUT
	DosingTotalizerVolume: REAL;
END_VAR

IF R2.RecipeStep[0].Started AND R2.RecipeStep[0].StartedTime = '' THEN
	//Update StartedTime
	R2.RecipeStep[0].StartedTime := MAIN.concatenatedHourMinuteString;
END_IF

// Start Block and HC Mode Selection
IF R2.RecipeStep[R2.R2STEPS].Started THEN
  R2.R2STEPS:= R2.R2STEPS+1;
 // R2.AbortRecipe:=FALSE;
  R2.ClearRecipe:=FALSE;
  R2.RecipeEnded:=FALSE;
END_IF  
 
// Check Process or JACKET SELECTION
IF R2.RecipeStep[0].HeatCoolModeSelection THEN
	R2.HeatCoolTemperatureControlType:=TRUE;
	R2.TemperatureControl:=REAL_TO_DINT(R2.ReactorMassTemperature);
ELSE
	R2.HeatCoolTemperatureControlType:=FALSE;	
	R2.TemperatureControl:=REAL_TO_DINT(R2.JacketOutletTemperature);
END_IF

 IF R2.RecipeStep[R2.R2STEPS].HeatcoolEnabled THEN
	R2.HeatCoolSetPoint:=R2.RecipeStep[R2.R2STEPS].HeatCoolSetpointExpression;		
	R2.RecipeStep[R2.R2STEPS].HeatCoolStarted :=TRUE;
	IF R2.RecipeStep[R2.R2STEPS].HeatCoolStartedTime = '' THEN
		R2.RecipeStep[R2.R2STEPS].HeatCoolStartedTime := Main.concatenatedHourMinuteString;
	END_IF
	R2.HeatCoolStatus:=TRUE;
	
		///Check for condition in step  
	 IF ABS(R2.TemperatureControl-R2.RecipeStep[R2.R2STEPS].HeatCoolSetpointExpression )<0.5 THEN
		R2.RecipeStep[R2.R2STEPS].HeatcoolEnded :=TRUE;	
		IF R2.RecipeStep[R2.R2STEPS].HeatCoolEndedTime = '' THEN
			R2.RecipeStep[R2.R2STEPS].HeatCoolEndedTime := Main.concatenatedHourMinuteString;
		END_IF
	 END_IF     	
 END_IF
	
////Recipe block for stirrer
IF R2.RecipeStep[R2.R2STEPS].StirrerEnabled THEN
	R2.StirrerSetPoint:=R2.RecipeStep[R2.R2STEPS].StirrerSetPointExpression;
	R2.StirrerStatus:=TRUE;	
    R2.RecipeStep[R2.R2STEPS].StirrerStarted:=TRUE;
	IF R2.RecipeStep[R2.R2STEPS].StirrerStartedTime = '' THEN
		R2.RecipeStep[R2.R2STEPS].StirrerStartedTime := Main.concatenatedHourMinuteString;
	END_IF
	
	///Check the Actual speed to end the step
      IF ABS(R2.StirrerCurrentSpeed- R2.RecipeStep[R2.R2STEPS].StirrerSetPointExpression)<8 THEN
		R2.RecipeStep[R2.R2STEPS].StirrerEnded:=TRUE;
		IF R2.RecipeStep[R2.R2STEPS].StirrerEndedTime = '' THEN
			R2.RecipeStep[R2.R2STEPS].StirrerEndedTime := Main.concatenatedHourMinuteString;
		END_IF
	  END_IF
	//Check the rpm TO switch off the vfd
	  IF R2.RecipeStep[R2.R2STEPS].StirrerSetPointExpression=0 THEN
		R2.StirrerStatus:=FALSE;	
	  END_IF///
  END_IF 


(*////Wait Block*)
IF R2.RecipeStep[R2.R2STEPS].WaitEnabled AND NOT R2.RecipeStep[R2STEPS].WaitEnded THEN
    R2.RecipeStep[R2.R2STEPS].WaitStarted:=TRUE;
	IF R2.RecipeStep[R2.R2STEPS].WaitStartedTime = '' THEN
		R2.RecipeStep[R2.R2STEPS].WaitStartedTime := Main.concatenatedHourMinuteString;
	END_IF
	R2.WaitTick:=R2.WaitTick+1;
	IF R2.WaitTick=100  THEN
		//Update the Second Tick
		R2.WaitSecondTick:=R2.WaitSecondTick+1;
		R2.WaitTick:=0;
	END_IF
		
	IF  R2.WaitSecondTick=60  THEN
		//Update the Minute Tick
		R2.WaitMinuteTick:=R2.WaitMinuteTick+1;
		R2.WaitSecondTick:=0;
	END_IF	

	//Update the Remaining Time
	remainingTimeCalculator(elapsedSeconds:= R2.WaitSecondTick, elapsedMinutes:= R2.WaitMinuteTick, givenDuration:= DINT_TO_INT(R2.RecipeStep[R2.R2STEPS].WaitDuration), 
							leftOverSeconds=> R2.RecipeStep[R2.R2STEPS].WaitRemainingSeconds, leftOverMinutes=> R2.RecipeStep[R2.R2STEPS].WaitRemainingMinutes);
	R2.RecipeStep[R2.R2STEPS].WaitRemainingTime := INT_TO_STRING(R2.RecipeStep[R2.R2STEPS].WaitRemainingMinutes);
	R2.RecipeStep[R2.R2STEPS].WaitRemainingTime := CONCAT(STR1:= R2.RecipeStep[R2.R2STEPS].WaitRemainingTime, STR2:= ':');
	R2.RecipeStep[R2.R2STEPS].WaitRemainingTime := CONCAT(STR1:= R2.RecipeStep[R2.R2STEPS].WaitRemainingTime, STR2:= INT_TO_STRING(R2.RecipeStep[R2.R2STEPS].WaitRemainingSeconds));
	
	(*///To write ended time*)
	IF ABS(R2.WaitMinuteTick -R2.RecipeStep[R2.R2STEPS].WaitDuration)=0 THEN
		R2.RecipeStep[R2.R2STEPS].WaitEnded:=TRUE;
		IF R2.RecipeStep[R2.R2STEPS].WaitEndedTime = '' THEN
			R2.RecipeStep[R2.R2STEPS].WaitEndedTime := Main.concatenatedHourMinuteString;
		END_IF
		R2.WaitTick:=0;
		R2.WaitSecondTick:=0;
		R2.WaitMinuteTick:=0;
	END_IF
END_IF
	
IF R2.RecipeStep[R2STEPS].DosingEnabled AND NOT R2.RecipeStep[R2STEPS].DosingEnded THEN
	R2.RecipeStep[R2STEPS].DosingStarted := TRUE;
	IF R2.RecipeStep[R2.R2STEPS].DosingStartedTime = '' THEN
		R2.RecipeStep[R2.R2STEPS].DosingStartedTime := Main.concatenatedHourMinuteString;
	END_IF
	//Update Totalized Volume
		IF  R2.DosingPumpStatus_1 THEN
			DosingTick:=DosingTick+1;
		END_IF
		   
	  IF DosingTick=100 THEN
		  DosingTotalizerVolume:=DosingTotalizerVolume+(R2.RecipeStep[R2STEPS].DosingRateSetpointExpression/2.7 * 0.045);	  
	  END_IF
	  
	  IF DosingTick>100 THEN
		  DosingTick:=0;
	  END_IF
	  
	IF DosingTotalizerVolume < R2.RecipeStep[R2STEPS].DosingMaxAmount THEN
		IF R2.DosingPumpStatus_1 THEN
			IF R2.TemperatureControl < R2.RecipeStep[R2STEPS].DosingStopTemp THEN
				R2.DosingPumpStatus_1 := TRUE;
				R2.DosingPumpSetPoint_1 := R2.RecipeStep[R2STEPS].DosingRateSetpointExpression;
			ELSE
				R2.DosingPumpStatus_1 := FALSE;
				R2.DosingPumpSetPoint_1 := 0;
			END_IF
		ELSE
			IF DosingTotalizerVolume = 0 AND R2.TemperatureControl > R2.RecipeStep[R2STEPS].DosingResumeTemp AND R2.TemperatureControl < R2.RecipeStep[R2STEPS].DosingStopTemp THEN
				//Logic for starting Dosing Pump First Time in a Recipe Step
				R2.DosingPumpStatus_1 := TRUE;
				R2.DosingPumpSetPoint_1 := R2.RecipeStep[R2STEPS].DosingRateSetpointExpression;
			END_IF
			
			IF R2.TemperatureControl < R2.RecipeStep[R2STEPS].DosingResumeTemp THEN
				R2.DosingPumpStatus_1 := TRUE;
				R2.DosingPumpSetPoint_1 := R2.RecipeStep[R2STEPS].DosingRateSetpointExpression;
			END_IF
		END_IF
	ELSE
		R2.DosingPumpStatus_1 := FALSE;
		R2.DosingPumpSetPoint_1 := 0;
		R2.RecipeStep[R2STEPS].DosingEnded := TRUE;
		IF R2.RecipeStep[R2.R2STEPS].DosingEndedTime = '' THEN
			R2.RecipeStep[R2.R2STEPS].DosingEndedTime := Main.concatenatedHourMinuteString;
		END_IF
		DosingTick := 0;
		DosingTotalizerVolume:=0;
	END_IF
END_IF

IF R2.R2STEPS>0 THEN 

(*//Step control block To increment to next step*)
 R2.TotalEnabledValue:=BOOL_TO_INT(R2.RecipeStep[R2.R2STEPS].HeatcoolEnabled)+BOOL_TO_INT(R2.RecipeStep[R2.R2STEPS].StirrerEnabled)+BOOL_TO_INT(R2.RecipeStep[R2.R2STEPS].WaitEnabled)+BOOL_TO_INT( R2.RecipeStep[R2.R2STEPS].DosingEnabled);
 R2.TotalEndedValue:=BOOL_TO_INT(R2.RecipeStep[R2.R2STEPS].HeatCoolEnded)+BOOL_TO_INT(R2.RecipeStep[R2.R2STEPS].StirrerEnded)+BOOL_TO_INT(R2.RecipeStep[R2.R2STEPS].WaitEnded)+BOOL_TO_INT( R2.RecipeStep[R2.R2STEPS].DosingEnded);

    IF (R2.TotalEnabledValue - R2.TotalEndedValue)=0 THEN 
		R2.R2STEPS:=R2.R2STEPS+1;
    END_IF
END_IF
  
 (* ///To End the Recipe**)
 IF  R2.NumberOfRecipeSteps = R2.R2STEPS THEN
	 R2.StirrerStatus:=FALSE;
	 R2.StirrerSetPoint:=0;
	 R2.HeatCoolStatus:=FALSE;
	 R2.HeatCoolSetPoint:=0;	
     R2.StepCompleted:=FALSE;	 
	 R2.RecipeEnded:=TRUE;
	 R2.RecipeStatus:=FALSE;
 END_IF
  
(* //TO ABORT RECIPE*)
AbortTrig(CLK:=R2.AbortRecipe,Q=>);
IF AbortTrig.Q THEN
	shutDownFB(GvlIdentifier := 'R2');
	AbortTrig.CLK := FALSE;
END_IF

END_PROGRAM

// ---- RecipeModules/RecipeModule_R3.TcPOU
PROGRAM RecipeModule_R3
VAR
	shutDownFB:Shutdown;
	remainingTimeCalculator : RemainingTimeCalculator;
	
	DosingTick: INT;
	AbortTrig:R_Trig;
END_VAR
VAR_INPUT
	DosingTotalizerVolume: REAL;
END_VAR

IF R3.RecipeStep[0].Started AND R3.RecipeStep[0].StartedTime = '' THEN
	//Update StartedTime
	R3.RecipeStep[0].StartedTime := MAIN.concatenatedHourMinuteString;
END_IF

// Start Block and HC Mode Selection
IF R3.RecipeStep[R3.R3STEPS].Started THEN
  R3.R3STEPS:= R3.R3STEPS+1;
 // R3.AbortRecipe:=FALSE;
  R3.ClearRecipe:=FALSE;
  R3.RecipeEnded:=FALSE;
END_IF  
 
// Check Process or JACKET SELECTION
IF R3.RecipeStep[0].HeatCoolModeSelection THEN
	R3.HeatCoolTemperatureControlType:=TRUE;
	R3.TemperatureControl:=REAL_TO_DINT(R3.ReactorMassTemperature);
ELSE
	R3.HeatCoolTemperatureControlType:=FALSE;	
	R3.TemperatureControl:=REAL_TO_DINT(R3.JacketOutletTemperature);
END_IF

 IF R3.RecipeStep[R3.R3STEPS].HeatcoolEnabled THEN
	R3.HeatCoolSetPoint:=R3.RecipeStep[R3.R3STEPS].HeatCoolSetpointExpression;		
	R3.RecipeStep[R3.R3STEPS].HeatCoolStarted :=TRUE;
	IF R3.RecipeStep[R3.R3STEPS].HeatCoolStartedTime = '' THEN
		R3.RecipeStep[R3.R3STEPS].HeatCoolStartedTime := Main.concatenatedHourMinuteString;
	END_IF
	R3.HeatCoolStatus:=TRUE;
	
		///Check for condition in step  
	 IF ABS(R3.TemperatureControl-R3.RecipeStep[R3.R3STEPS].HeatCoolSetpointExpression )<0.5 THEN
		R3.RecipeStep[R3.R3STEPS].HeatcoolEnded :=TRUE;	
		IF R3.RecipeStep[R3.R3STEPS].HeatCoolEndedTime = '' THEN
			R3.RecipeStep[R3.R3STEPS].HeatCoolEndedTime := Main.concatenatedHourMinuteString;
		END_IF
	 END_IF     	
 END_IF
	
////Recipe block for stirrer
IF R3.RecipeStep[R3.R3STEPS].StirrerEnabled THEN
	R3.StirrerSetPoint:=R3.RecipeStep[R3.R3STEPS].StirrerSetPointExpression;
	R3.StirrerStatus:=TRUE;	
    R3.RecipeStep[R3.R3STEPS].StirrerStarted:=TRUE;
	IF R3.RecipeStep[R3.R3STEPS].StirrerStartedTime = '' THEN
		R3.RecipeStep[R3.R3STEPS].StirrerStartedTime := Main.concatenatedHourMinuteString;
	END_IF
	
	///Check the Actual speed to end the step
      IF ABS(R3.StirrerCurrentSpeed- R3.RecipeStep[R3.R3STEPS].StirrerSetPointExpression)<8 THEN
		R3.RecipeStep[R3.R3STEPS].StirrerEnded:=TRUE;
		IF R3.RecipeStep[R3.R3STEPS].StirrerEndedTime = '' THEN
			R3.RecipeStep[R3.R3STEPS].StirrerEndedTime := Main.concatenatedHourMinuteString;
		END_IF
	  END_IF
	//Check the rpm TO switch off the vfd
	  IF R3.RecipeStep[R3.R3STEPS].StirrerSetPointExpression=0 THEN
		R3.StirrerStatus:=FALSE;	
	  END_IF///
  END_IF 


(*////Wait Block*)
IF R3.RecipeStep[R3.R3STEPS].WaitEnabled AND NOT R3.RecipeStep[R3STEPS].WaitEnded THEN
    R3.RecipeStep[R3.R3STEPS].WaitStarted:=TRUE;
	IF R3.RecipeStep[R3.R3STEPS].WaitStartedTime = '' THEN
		R3.RecipeStep[R3.R3STEPS].WaitStartedTime := Main.concatenatedHourMinuteString;
	END_IF
	R3.WaitTick:=R3.WaitTick+1;
	IF R3.WaitTick=100  THEN
		//Update the Second Tick
		R3.WaitSecondTick:=R3.WaitSecondTick+1;
		R3.WaitTick:=0;
	END_IF
		
	IF  R3.WaitSecondTick=60  THEN
		//Update the Minute Tick
		R3.WaitMinuteTick:=R3.WaitMinuteTick+1;
		R3.WaitSecondTick:=0;
	END_IF	

	//Update the Remaining Time
	remainingTimeCalculator(elapsedSeconds:= R3.WaitSecondTick, elapsedMinutes:= R3.WaitMinuteTick, givenDuration:= DINT_TO_INT(R3.RecipeStep[R3.R3STEPS].WaitDuration), 
							leftOverSeconds=> R3.RecipeStep[R3.R3STEPS].WaitRemainingSeconds, leftOverMinutes=> R3.RecipeStep[R3.R3STEPS].WaitRemainingMinutes);
	R3.RecipeStep[R3.R3STEPS].WaitRemainingTime := INT_TO_STRING(R3.RecipeStep[R3.R3STEPS].WaitRemainingMinutes);
	R3.RecipeStep[R3.R3STEPS].WaitRemainingTime := CONCAT(STR1:= R3.RecipeStep[R3.R3STEPS].WaitRemainingTime, STR2:= ':');
	R3.RecipeStep[R3.R3STEPS].WaitRemainingTime := CONCAT(STR1:= R3.RecipeStep[R3.R3STEPS].WaitRemainingTime, STR2:= INT_TO_STRING(R3.RecipeStep[R3.R3STEPS].WaitRemainingSeconds));
	
	(*///To write ended time*)
	IF ABS(R3.WaitMinuteTick -R3.RecipeStep[R3.R3STEPS].WaitDuration)=0 THEN
		R3.RecipeStep[R3.R3STEPS].WaitEnded:=TRUE;
		IF R3.RecipeStep[R3.R3STEPS].WaitEndedTime = '' THEN
			R3.RecipeStep[R3.R3STEPS].WaitEndedTime := Main.concatenatedHourMinuteString;
		END_IF
		R3.WaitTick:=0;
		R3.WaitSecondTick:=0;
		R3.WaitMinuteTick:=0;
	END_IF
END_IF
	
IF R3.RecipeStep[R3STEPS].DosingEnabled AND NOT R3.RecipeStep[R3STEPS].DosingEnded THEN
	R3.RecipeStep[R3STEPS].DosingStarted := TRUE;
	IF R3.RecipeStep[R3.R3STEPS].DosingStartedTime = '' THEN
		R3.RecipeStep[R3.R3STEPS].DosingStartedTime := Main.concatenatedHourMinuteString;
	END_IF
	//Update Totalized Volume
		IF  R3.DosingPumpStatus_1 THEN
			DosingTick:=DosingTick+1;
		END_IF
		   
	  IF DosingTick=100 THEN
		  DosingTotalizerVolume:=DosingTotalizerVolume+(R3.RecipeStep[R3STEPS].DosingRateSetpointExpression/2.7 * 0.045);	  
	  END_IF
	  
	  IF DosingTick>100 THEN
		  DosingTick:=0;
	  END_IF
	  
	IF DosingTotalizerVolume < R3.RecipeStep[R3STEPS].DosingMaxAmount THEN
		IF R3.DosingPumpStatus_1 THEN
			IF R3.TemperatureControl < R3.RecipeStep[R3STEPS].DosingStopTemp THEN
				R3.DosingPumpStatus_1 := TRUE;
				R3.DosingPumpSetPoint_1 := R3.RecipeStep[R3STEPS].DosingRateSetpointExpression;
			ELSE
				R3.DosingPumpStatus_1 := FALSE;
				R3.DosingPumpSetPoint_1 := 0;
			END_IF
		ELSE
			IF DosingTotalizerVolume = 0 AND R3.TemperatureControl > R3.RecipeStep[R3STEPS].DosingResumeTemp AND R3.TemperatureControl < R3.RecipeStep[R3STEPS].DosingStopTemp THEN
				//Logic for starting Dosing Pump First Time in a Recipe Step
				R3.DosingPumpStatus_1 := TRUE;
				R3.DosingPumpSetPoint_1 := R3.RecipeStep[R3STEPS].DosingRateSetpointExpression;
			END_IF
			
			IF R3.TemperatureControl < R3.RecipeStep[R3STEPS].DosingResumeTemp THEN
				R3.DosingPumpStatus_1 := TRUE;
				R3.DosingPumpSetPoint_1 := R3.RecipeStep[R3STEPS].DosingRateSetpointExpression;
			END_IF
		END_IF
	ELSE
		R3.DosingPumpStatus_1 := FALSE;
		R3.DosingPumpSetPoint_1 := 0;
		R3.RecipeStep[R3STEPS].DosingEnded := TRUE;
		IF R3.RecipeStep[R3.R3STEPS].DosingEndedTime = '' THEN
			R3.RecipeStep[R3.R3STEPS].DosingEndedTime := Main.concatenatedHourMinuteString;
		END_IF
		DosingTick := 0;
		DosingTotalizerVolume:=0;
	END_IF
END_IF

IF R3.R3STEPS>0 THEN 

(*//Step control block To increment to next step*)
 R3.TotalEnabledValue:=BOOL_TO_INT(R3.RecipeStep[R3.R3STEPS].HeatcoolEnabled)+BOOL_TO_INT(R3.RecipeStep[R3.R3STEPS].StirrerEnabled)+BOOL_TO_INT(R3.RecipeStep[R3.R3STEPS].WaitEnabled)+BOOL_TO_INT( R3.RecipeStep[R3.R3STEPS].DosingEnabled);
 R3.TotalEndedValue:=BOOL_TO_INT(R3.RecipeStep[R3.R3STEPS].HeatCoolEnded)+BOOL_TO_INT(R3.RecipeStep[R3.R3STEPS].StirrerEnded)+BOOL_TO_INT(R3.RecipeStep[R3.R3STEPS].WaitEnded)+BOOL_TO_INT( R3.RecipeStep[R3.R3STEPS].DosingEnded);

    IF (R3.TotalEnabledValue - R3.TotalEndedValue)=0 THEN 
		R3.R3STEPS:=R3.R3STEPS+1;
    END_IF
END_IF
  
 (* ///To End the Recipe**)
 IF  R3.NumberOfRecipeSteps = R3.R3STEPS THEN
	 R3.StirrerStatus:=FALSE;
	 R3.StirrerSetPoint:=0;
	 R3.HeatCoolStatus:=FALSE;
	 R3.HeatCoolSetPoint:=0;	
     R3.StepCompleted:=FALSE;	 
	 R3.RecipeEnded:=TRUE;
	 R3.RecipeStatus:=FALSE;
 END_IF
  
(* //TO ABORT RECIPE*)
AbortTrig(CLK:=R3.AbortRecipe,Q=>);
IF AbortTrig.Q THEN
	shutDownFB(GvlIdentifier := 'R3');
	AbortTrig.CLK := FALSE;
END_IF

END_PROGRAM

// ---- RecipeModules/RecipeModule_R4.TcPOU
PROGRAM RecipeModule_R4
VAR
	shutDownFB:Shutdown;
	remainingTimeCalculator : RemainingTimeCalculator;
	
	DosingTick: INT;
	AbortTrig:R_Trig;
END_VAR
VAR_INPUT
	DosingTotalizerVolume: REAL;
END_VAR

IF R4.RecipeStep[0].Started AND R4.RecipeStep[0].StartedTime = '' THEN
	//Update StartedTime
	R4.RecipeStep[0].StartedTime := MAIN.concatenatedHourMinuteString;
END_IF

// Start Block and HC Mode Selection
IF R4.RecipeStep[R4.R4STEPS].Started THEN
  R4.R4STEPS:= R4.R4STEPS+1;
 // R4.AbortRecipe:=FALSE;
  R4.ClearRecipe:=FALSE;
  R4.RecipeEnded:=FALSE;
END_IF  
 
// Check Process or JACKET SELECTION
IF R4.RecipeStep[0].HeatCoolModeSelection THEN
	R4.HeatCoolTemperatureControlType:=TRUE;
	R4.TemperatureControl:=REAL_TO_DINT(R4.ReactorMassTemperature);
ELSE
	R4.HeatCoolTemperatureControlType:=FALSE;	
	R4.TemperatureControl:=REAL_TO_DINT(R4.JacketOutletTemperature);
END_IF

 IF R4.RecipeStep[R4.R4STEPS].HeatcoolEnabled THEN
	R4.HeatCoolSetPoint:=R4.RecipeStep[R4.R4STEPS].HeatCoolSetpointExpression;		
	R4.RecipeStep[R4.R4STEPS].HeatCoolStarted :=TRUE;
	IF R4.RecipeStep[R4.R4STEPS].HeatCoolStartedTime = '' THEN
		R4.RecipeStep[R4.R4STEPS].HeatCoolStartedTime := Main.concatenatedHourMinuteString;
	END_IF
	R4.HeatCoolStatus:=TRUE;
	
		///Check for condition in step  
	 IF ABS(R4.TemperatureControl-R4.RecipeStep[R4.R4STEPS].HeatCoolSetpointExpression )<0.5 THEN
		R4.RecipeStep[R4.R4STEPS].HeatcoolEnded :=TRUE;	
		IF R4.RecipeStep[R4.R4STEPS].HeatCoolEndedTime = '' THEN
			R4.RecipeStep[R4.R4STEPS].HeatCoolEndedTime := Main.concatenatedHourMinuteString;
		END_IF
	 END_IF     	
 END_IF
	
////Recipe block for stirrer
IF R4.RecipeStep[R4.R4STEPS].StirrerEnabled THEN
	R4.StirrerSetPoint:=R4.RecipeStep[R4.R4STEPS].StirrerSetPointExpression;
	R4.StirrerStatus:=TRUE;	
    R4.RecipeStep[R4.R4STEPS].StirrerStarted:=TRUE;
	IF R4.RecipeStep[R4.R4STEPS].StirrerStartedTime = '' THEN
		R4.RecipeStep[R4.R4STEPS].StirrerStartedTime := Main.concatenatedHourMinuteString;
	END_IF
	
	///Check the Actual speed to end the step
      IF ABS(R4.StirrerCurrentSpeed- R4.RecipeStep[R4.R4STEPS].StirrerSetPointExpression)<8 THEN
		R4.RecipeStep[R4.R4STEPS].StirrerEnded:=TRUE;
		IF R4.RecipeStep[R4.R4STEPS].StirrerEndedTime = '' THEN
			R4.RecipeStep[R4.R4STEPS].StirrerEndedTime := Main.concatenatedHourMinuteString;
		END_IF
	  END_IF
	//Check the rpm TO switch off the vfd
	  IF R4.RecipeStep[R4.R4STEPS].StirrerSetPointExpression=0 THEN
		R4.StirrerStatus:=FALSE;	
	  END_IF///
  END_IF 


(*////Wait Block*)
IF R4.RecipeStep[R4.R4STEPS].WaitEnabled AND NOT R4.RecipeStep[R4STEPS].WaitEnded THEN
    R4.RecipeStep[R4.R4STEPS].WaitStarted:=TRUE;
	IF R4.RecipeStep[R4.R4STEPS].WaitStartedTime = '' THEN
		R4.RecipeStep[R4.R4STEPS].WaitStartedTime := Main.concatenatedHourMinuteString;
	END_IF
	R4.WaitTick:=R4.WaitTick+1;
	IF R4.WaitTick=100  THEN
		//Update the Second Tick
		R4.WaitSecondTick:=R4.WaitSecondTick+1;
		R4.WaitTick:=0;
	END_IF
		
	IF  R4.WaitSecondTick=60  THEN
		//Update the Minute Tick
		R4.WaitMinuteTick:=R4.WaitMinuteTick+1;
		R4.WaitSecondTick:=0;
	END_IF	

	//Update the Remaining Time
	remainingTimeCalculator(elapsedSeconds:= R4.WaitSecondTick, elapsedMinutes:= R4.WaitMinuteTick, givenDuration:= DINT_TO_INT(R4.RecipeStep[R4.R4STEPS].WaitDuration), 
							leftOverSeconds=> R4.RecipeStep[R4.R4STEPS].WaitRemainingSeconds, leftOverMinutes=> R4.RecipeStep[R4.R4STEPS].WaitRemainingMinutes);
	R4.RecipeStep[R4.R4STEPS].WaitRemainingTime := INT_TO_STRING(R4.RecipeStep[R4.R4STEPS].WaitRemainingMinutes);
	R4.RecipeStep[R4.R4STEPS].WaitRemainingTime := CONCAT(STR1:= R4.RecipeStep[R4.R4STEPS].WaitRemainingTime, STR2:= ':');
	R4.RecipeStep[R4.R4STEPS].WaitRemainingTime := CONCAT(STR1:= R4.RecipeStep[R4.R4STEPS].WaitRemainingTime, STR2:= INT_TO_STRING(R4.RecipeStep[R4.R4STEPS].WaitRemainingSeconds));
	
	(*///To write ended time*)
	IF ABS(R4.WaitMinuteTick -R4.RecipeStep[R4.R4STEPS].WaitDuration)=0 THEN
		R4.RecipeStep[R4.R4STEPS].WaitEnded:=TRUE;
		IF R4.RecipeStep[R4.R4STEPS].WaitEndedTime = '' THEN
			R4.RecipeStep[R4.R4STEPS].WaitEndedTime := Main.concatenatedHourMinuteString;
		END_IF
		R4.WaitTick:=0;
		R4.WaitSecondTick:=0;
		R4.WaitMinuteTick:=0;
	END_IF
END_IF
	
IF R4.RecipeStep[R4STEPS].DosingEnabled AND NOT R4.RecipeStep[R4STEPS].DosingEnded THEN
	R4.RecipeStep[R4STEPS].DosingStarted := TRUE;
	IF R4.RecipeStep[R4.R4STEPS].DosingStartedTime = '' THEN
		R4.RecipeStep[R4.R4STEPS].DosingStartedTime := Main.concatenatedHourMinuteString;
	END_IF
	//Update Totalized Volume
		IF  R4.DosingPumpStatus_1 THEN
			DosingTick:=DosingTick+1;
		END_IF
		   
	  IF DosingTick=100 THEN
		  DosingTotalizerVolume:=DosingTotalizerVolume+(R4.RecipeStep[R4STEPS].DosingRateSetpointExpression/2.7 * 0.045);	  
	  END_IF
	  
	  IF DosingTick>100 THEN
		  DosingTick:=0;
	  END_IF
	  
	IF DosingTotalizerVolume < R4.RecipeStep[R4STEPS].DosingMaxAmount THEN
		IF R4.DosingPumpStatus_1 THEN
			IF R4.TemperatureControl < R4.RecipeStep[R4STEPS].DosingStopTemp THEN
				R4.DosingPumpStatus_1 := TRUE;
				R4.DosingPumpSetPoint_1 := R4.RecipeStep[R4STEPS].DosingRateSetpointExpression;
			ELSE
				R4.DosingPumpStatus_1 := FALSE;
				R4.DosingPumpSetPoint_1 := 0;
			END_IF
		ELSE
			IF DosingTotalizerVolume = 0 AND R4.TemperatureControl > R4.RecipeStep[R4STEPS].DosingResumeTemp AND R4.TemperatureControl < R4.RecipeStep[R4STEPS].DosingStopTemp THEN
				//Logic for starting Dosing Pump First Time in a Recipe Step
				R4.DosingPumpStatus_1 := TRUE;
				R4.DosingPumpSetPoint_1 := R4.RecipeStep[R4STEPS].DosingRateSetpointExpression;
			END_IF
			
			IF R4.TemperatureControl < R4.RecipeStep[R4STEPS].DosingResumeTemp THEN
				R4.DosingPumpStatus_1 := TRUE;
				R4.DosingPumpSetPoint_1 := R4.RecipeStep[R4STEPS].DosingRateSetpointExpression;
			END_IF
		END_IF
	ELSE
		R4.DosingPumpStatus_1 := FALSE;
		R4.DosingPumpSetPoint_1 := 0;
		R4.RecipeStep[R4STEPS].DosingEnded := TRUE;
		IF R4.RecipeStep[R4.R4STEPS].DosingEndedTime = '' THEN
			R4.RecipeStep[R4.R4STEPS].DosingEndedTime := Main.concatenatedHourMinuteString;
		END_IF
		DosingTick := 0;
		DosingTotalizerVolume:=0;
	END_IF
END_IF

IF R4.R4STEPS>0 THEN 

(*//Step control block To increment to next step*)
 R4.TotalEnabledValue:=BOOL_TO_INT(R4.RecipeStep[R4.R4STEPS].HeatcoolEnabled)+BOOL_TO_INT(R4.RecipeStep[R4.R4STEPS].StirrerEnabled)+BOOL_TO_INT(R4.RecipeStep[R4.R4STEPS].WaitEnabled)+BOOL_TO_INT( R4.RecipeStep[R4.R4STEPS].DosingEnabled);
 R4.TotalEndedValue:=BOOL_TO_INT(R4.RecipeStep[R4.R4STEPS].HeatCoolEnded)+BOOL_TO_INT(R4.RecipeStep[R4.R4STEPS].StirrerEnded)+BOOL_TO_INT(R4.RecipeStep[R4.R4STEPS].WaitEnded)+BOOL_TO_INT( R4.RecipeStep[R4.R4STEPS].DosingEnded);

    IF (R4.TotalEnabledValue - R4.TotalEndedValue)=0 THEN 
		R4.R4STEPS:=R4.R4STEPS+1;
    END_IF
END_IF
  
 (* ///To End the Recipe**)
 IF  R4.NumberOfRecipeSteps = R4.R4STEPS THEN
	 R4.StirrerStatus:=FALSE;
	 R4.StirrerSetPoint:=0;
	 R4.HeatCoolStatus:=FALSE;
	 R4.HeatCoolSetPoint:=0;	
     R4.StepCompleted:=FALSE;	 
	 R4.RecipeEnded:=TRUE;
	 R4.RecipeStatus:=FALSE;
 END_IF
  
(* //TO ABORT RECIPE*)
AbortTrig(CLK:=R4.AbortRecipe,Q=>);
IF AbortTrig.Q THEN
	shutDownFB(GvlIdentifier := 'R4');
	AbortTrig.CLK := FALSE;
END_IF

END_PROGRAM

// ---- RecipeModules/RecipeModule_R5.TcPOU
PROGRAM RecipeModule_R5
VAR
	shutDownFB:Shutdown;
	remainingTimeCalculator : RemainingTimeCalculator;
	
	DosingTick: INT;
	AbortTrig:R_Trig;
END_VAR
VAR_INPUT
	DosingTotalizerVolume: REAL;
END_VAR

IF R5.RecipeStep[0].Started AND R5.RecipeStep[0].StartedTime = '' THEN
	//Update StartedTime
	R5.RecipeStep[0].StartedTime := MAIN.concatenatedHourMinuteString;
END_IF

// Start Block and HC Mode Selection
IF R5.RecipeStep[R5.R5STEPS].Started THEN
  R5.R5STEPS:= R5.R5STEPS+1;
 // R5.AbortRecipe:=FALSE;
  R5.ClearRecipe:=FALSE;
  R5.RecipeEnded:=FALSE;
END_IF  
 
// Check Process or JACKET SELECTION
IF R5.RecipeStep[0].HeatCoolModeSelection THEN
	R5.HeatCoolTemperatureControlType:=TRUE;
	R5.TemperatureControl:=REAL_TO_DINT(R5.ReactorMassTemperature);
ELSE
	R5.HeatCoolTemperatureControlType:=FALSE;	
	R5.TemperatureControl:=REAL_TO_DINT(R5.JacketOutletTemperature);
END_IF

 IF R5.RecipeStep[R5.R5STEPS].HeatcoolEnabled THEN
	R5.HeatCoolSetPoint:=R5.RecipeStep[R5.R5STEPS].HeatCoolSetpointExpression;		
	R5.RecipeStep[R5.R5STEPS].HeatCoolStarted :=TRUE;
	IF R5.RecipeStep[R5.R5STEPS].HeatCoolStartedTime = '' THEN
		R5.RecipeStep[R5.R5STEPS].HeatCoolStartedTime := Main.concatenatedHourMinuteString;
	END_IF
	R5.HeatCoolStatus:=TRUE;
	
		///Check for condition in step  
	 IF ABS(R5.TemperatureControl-R5.RecipeStep[R5.R5STEPS].HeatCoolSetpointExpression )<0.5 THEN
		R5.RecipeStep[R5.R5STEPS].HeatcoolEnded :=TRUE;	
		IF R5.RecipeStep[R5.R5STEPS].HeatCoolEndedTime = '' THEN
			R5.RecipeStep[R5.R5STEPS].HeatCoolEndedTime := Main.concatenatedHourMinuteString;
		END_IF
	 END_IF     	
 END_IF
	
////Recipe block for stirrer
IF R5.RecipeStep[R5.R5STEPS].StirrerEnabled THEN
	R5.StirrerSetPoint:=R5.RecipeStep[R5.R5STEPS].StirrerSetPointExpression;
	R5.StirrerStatus:=TRUE;	
    R5.RecipeStep[R5.R5STEPS].StirrerStarted:=TRUE;
	IF R5.RecipeStep[R5.R5STEPS].StirrerStartedTime = '' THEN
		R5.RecipeStep[R5.R5STEPS].StirrerStartedTime := Main.concatenatedHourMinuteString;
	END_IF
	
	///Check the Actual speed to end the step
      IF ABS(R5.StirrerCurrentSpeed- R5.RecipeStep[R5.R5STEPS].StirrerSetPointExpression)<8 THEN
		R5.RecipeStep[R5.R5STEPS].StirrerEnded:=TRUE;
		IF R5.RecipeStep[R5.R5STEPS].StirrerEndedTime = '' THEN
			R5.RecipeStep[R5.R5STEPS].StirrerEndedTime := Main.concatenatedHourMinuteString;
		END_IF
	  END_IF
	//Check the rpm TO switch off the vfd
	  IF R5.RecipeStep[R5.R5STEPS].StirrerSetPointExpression=0 THEN
		R5.StirrerStatus:=FALSE;	
	  END_IF///
  END_IF 


(*////Wait Block*)
IF R5.RecipeStep[R5.R5STEPS].WaitEnabled AND NOT R5.RecipeStep[R5STEPS].WaitEnded THEN
    R5.RecipeStep[R5.R5STEPS].WaitStarted:=TRUE;
	IF R5.RecipeStep[R5.R5STEPS].WaitStartedTime = '' THEN
		R5.RecipeStep[R5.R5STEPS].WaitStartedTime := Main.concatenatedHourMinuteString;
	END_IF
	R5.WaitTick:=R5.WaitTick+1;
	IF R5.WaitTick=100  THEN
		//Update the Second Tick
		R5.WaitSecondTick:=R5.WaitSecondTick+1;
		R5.WaitTick:=0;
	END_IF
		
	IF  R5.WaitSecondTick=60  THEN
		//Update the Minute Tick
		R5.WaitMinuteTick:=R5.WaitMinuteTick+1;
		R5.WaitSecondTick:=0;
	END_IF	

	//Update the Remaining Time
	remainingTimeCalculator(elapsedSeconds:= R5.WaitSecondTick, elapsedMinutes:= R5.WaitMinuteTick, givenDuration:= DINT_TO_INT(R5.RecipeStep[R5.R5STEPS].WaitDuration), 
							leftOverSeconds=> R5.RecipeStep[R5.R5STEPS].WaitRemainingSeconds, leftOverMinutes=> R5.RecipeStep[R5.R5STEPS].WaitRemainingMinutes);
	R5.RecipeStep[R5.R5STEPS].WaitRemainingTime := INT_TO_STRING(R5.RecipeStep[R5.R5STEPS].WaitRemainingMinutes);
	R5.RecipeStep[R5.R5STEPS].WaitRemainingTime := CONCAT(STR1:= R5.RecipeStep[R5.R5STEPS].WaitRemainingTime, STR2:= ':');
	R5.RecipeStep[R5.R5STEPS].WaitRemainingTime := CONCAT(STR1:= R5.RecipeStep[R5.R5STEPS].WaitRemainingTime, STR2:= INT_TO_STRING(R5.RecipeStep[R5.R5STEPS].WaitRemainingSeconds));
	
	(*///To write ended time*)
	IF ABS(R5.WaitMinuteTick -R5.RecipeStep[R5.R5STEPS].WaitDuration)=0 THEN
		R5.RecipeStep[R5.R5STEPS].WaitEnded:=TRUE;
		IF R5.RecipeStep[R5.R5STEPS].WaitEndedTime = '' THEN
			R5.RecipeStep[R5.R5STEPS].WaitEndedTime := Main.concatenatedHourMinuteString;
		END_IF
		R5.WaitTick:=0;
		R5.WaitSecondTick:=0;
		R5.WaitMinuteTick:=0;
	END_IF
END_IF
	
IF R5.RecipeStep[R5STEPS].DosingEnabled AND NOT R5.RecipeStep[R5STEPS].DosingEnded THEN
	R5.RecipeStep[R5STEPS].DosingStarted := TRUE;
	IF R5.RecipeStep[R5.R5STEPS].DosingStartedTime = '' THEN
		R5.RecipeStep[R5.R5STEPS].DosingStartedTime := Main.concatenatedHourMinuteString;
	END_IF
	//Update Totalized Volume
		IF  R5.DosingPumpStatus_1 THEN
			DosingTick:=DosingTick+1;
		END_IF
		   
	  IF DosingTick=100 THEN
		  DosingTotalizerVolume:=DosingTotalizerVolume+(R5.RecipeStep[R5STEPS].DosingRateSetpointExpression/2.7 * 0.045);	  
	  END_IF
	  
	  IF DosingTick>100 THEN
		  DosingTick:=0;
	  END_IF
	  
	IF DosingTotalizerVolume < R5.RecipeStep[R5STEPS].DosingMaxAmount THEN
		IF R5.DosingPumpStatus_1 THEN
			IF R5.TemperatureControl < R5.RecipeStep[R5STEPS].DosingStopTemp THEN
				R5.DosingPumpStatus_1 := TRUE;
				R5.DosingPumpSetPoint_1 := R5.RecipeStep[R5STEPS].DosingRateSetpointExpression;
			ELSE
				R5.DosingPumpStatus_1 := FALSE;
				R5.DosingPumpSetPoint_1 := 0;
			END_IF
		ELSE
			IF DosingTotalizerVolume = 0 AND R5.TemperatureControl > R5.RecipeStep[R5STEPS].DosingResumeTemp AND R5.TemperatureControl < R5.RecipeStep[R5STEPS].DosingStopTemp THEN
				//Logic for starting Dosing Pump First Time in a Recipe Step
				R5.DosingPumpStatus_1 := TRUE;
				R5.DosingPumpSetPoint_1 := R5.RecipeStep[R5STEPS].DosingRateSetpointExpression;
			END_IF
			
			IF R5.TemperatureControl < R5.RecipeStep[R5STEPS].DosingResumeTemp THEN
				R5.DosingPumpStatus_1 := TRUE;
				R5.DosingPumpSetPoint_1 := R5.RecipeStep[R5STEPS].DosingRateSetpointExpression;
			END_IF
		END_IF
	ELSE
		R5.DosingPumpStatus_1 := FALSE;
		R5.DosingPumpSetPoint_1 := 0;
		R5.RecipeStep[R5STEPS].DosingEnded := TRUE;
		IF R5.RecipeStep[R5.R5STEPS].DosingEndedTime = '' THEN
			R5.RecipeStep[R5.R5STEPS].DosingEndedTime := Main.concatenatedHourMinuteString;
		END_IF
		DosingTick := 0;
		DosingTotalizerVolume:=0;
	END_IF
END_IF

IF R5.R5STEPS>0 THEN 

(*//Step control block To increment to next step*)
 R5.TotalEnabledValue:=BOOL_TO_INT(R5.RecipeStep[R5.R5STEPS].HeatcoolEnabled)+BOOL_TO_INT(R5.RecipeStep[R5.R5STEPS].StirrerEnabled)+BOOL_TO_INT(R5.RecipeStep[R5.R5STEPS].WaitEnabled)+BOOL_TO_INT( R5.RecipeStep[R5.R5STEPS].DosingEnabled);
 R5.TotalEndedValue:=BOOL_TO_INT(R5.RecipeStep[R5.R5STEPS].HeatCoolEnded)+BOOL_TO_INT(R5.RecipeStep[R5.R5STEPS].StirrerEnded)+BOOL_TO_INT(R5.RecipeStep[R5.R5STEPS].WaitEnded)+BOOL_TO_INT( R5.RecipeStep[R5.R5STEPS].DosingEnded);

    IF (R5.TotalEnabledValue - R5.TotalEndedValue)=0 THEN 
		R5.R5STEPS:=R5.R5STEPS+1;
    END_IF
END_IF
  
 (* ///To End the Recipe**)
 IF  R5.NumberOfRecipeSteps = R5.R5STEPS THEN
	 R5.StirrerStatus:=FALSE;
	 R5.StirrerSetPoint:=0;
	 R5.HeatCoolStatus:=FALSE;
	 R5.HeatCoolSetPoint:=0;	
     R5.StepCompleted:=FALSE;	 
	 R5.RecipeEnded:=TRUE;
	 R5.RecipeStatus:=FALSE;
 END_IF
  
(* //TO ABORT RECIPE*)
AbortTrig(CLK:=R5.AbortRecipe,Q=>);
IF AbortTrig.Q THEN
	shutDownFB(GvlIdentifier := 'R5');
	AbortTrig.CLK := FALSE;
END_IF

END_PROGRAM

// ---- RecipeModules/RecipeModule_R6.TcPOU
PROGRAM RecipeModule_R6
VAR
	shutDownFB:Shutdown;
	remainingTimeCalculator : RemainingTimeCalculator;
	
	DosingTick: INT;
	AbortTrig:R_Trig;
END_VAR
VAR_INPUT
	DosingTotalizerVolume: REAL;
END_VAR

IF R6.RecipeStep[0].Started AND R6.RecipeStep[0].StartedTime = '' THEN
	//Update StartedTime
	R6.RecipeStep[0].StartedTime := MAIN.concatenatedHourMinuteString;
END_IF

// Start Block and HC Mode Selection
IF R6.RecipeStep[R6.R6STEPS].Started THEN
  R6.R6STEPS:= R6.R6STEPS+1;
 // R6.AbortRecipe:=FALSE;
  R6.ClearRecipe:=FALSE;
  R6.RecipeEnded:=FALSE;
END_IF  
 
// Check Process or JACKET SELECTION
IF R6.RecipeStep[0].HeatCoolModeSelection THEN
	R6.HeatCoolTemperatureControlType:=TRUE;
	R6.TemperatureControl:=REAL_TO_DINT(R6.ReactorMassTemperature);
ELSE
	R6.HeatCoolTemperatureControlType:=FALSE;	
	R6.TemperatureControl:=REAL_TO_DINT(R6.JacketOutletTemperature);
END_IF

 IF R6.RecipeStep[R6.R6STEPS].HeatcoolEnabled THEN
	R6.HeatCoolSetPoint:=R6.RecipeStep[R6.R6STEPS].HeatCoolSetpointExpression;		
	R6.RecipeStep[R6.R6STEPS].HeatCoolStarted :=TRUE;
	IF R6.RecipeStep[R6.R6STEPS].HeatCoolStartedTime = '' THEN
		R6.RecipeStep[R6.R6STEPS].HeatCoolStartedTime := Main.concatenatedHourMinuteString;
	END_IF
	R6.HeatCoolStatus:=TRUE;
	
		///Check for condition in step  
	 IF ABS(R6.TemperatureControl-R6.RecipeStep[R6.R6STEPS].HeatCoolSetpointExpression )<0.5 THEN
		R6.RecipeStep[R6.R6STEPS].HeatcoolEnded :=TRUE;	
		IF R6.RecipeStep[R6.R6STEPS].HeatCoolEndedTime = '' THEN
			R6.RecipeStep[R6.R6STEPS].HeatCoolEndedTime := Main.concatenatedHourMinuteString;
		END_IF
	 END_IF     	
 END_IF
	
////Recipe block for stirrer
IF R6.RecipeStep[R6.R6STEPS].StirrerEnabled THEN
	R6.StirrerSetPoint:=R6.RecipeStep[R6.R6STEPS].StirrerSetPointExpression;
	R6.StirrerStatus:=TRUE;	
    R6.RecipeStep[R6.R6STEPS].StirrerStarted:=TRUE;
	IF R6.RecipeStep[R6.R6STEPS].StirrerStartedTime = '' THEN
		R6.RecipeStep[R6.R6STEPS].StirrerStartedTime := Main.concatenatedHourMinuteString;
	END_IF
	
	///Check the Actual speed to end the step
      IF ABS(R6.StirrerCurrentSpeed- R6.RecipeStep[R6.R6STEPS].StirrerSetPointExpression)<8 THEN
		R6.RecipeStep[R6.R6STEPS].StirrerEnded:=TRUE;
		IF R6.RecipeStep[R6.R6STEPS].StirrerEndedTime = '' THEN
			R6.RecipeStep[R6.R6STEPS].StirrerEndedTime := Main.concatenatedHourMinuteString;
		END_IF
	  END_IF
	//Check the rpm TO switch off the vfd
	  IF R6.RecipeStep[R6.R6STEPS].StirrerSetPointExpression=0 THEN
		R6.StirrerStatus:=FALSE;	
	  END_IF///
  END_IF 


(*////Wait Block*)
IF R6.RecipeStep[R6.R6STEPS].WaitEnabled AND NOT R6.RecipeStep[R6STEPS].WaitEnded THEN
    R6.RecipeStep[R6.R6STEPS].WaitStarted:=TRUE;
	IF R6.RecipeStep[R6.R6STEPS].WaitStartedTime = '' THEN
		R6.RecipeStep[R6.R6STEPS].WaitStartedTime := Main.concatenatedHourMinuteString;
	END_IF
	R6.WaitTick:=R6.WaitTick+1;
	IF R6.WaitTick=100  THEN
		//Update the Second Tick
		R6.WaitSecondTick:=R6.WaitSecondTick+1;
		R6.WaitTick:=0;
	END_IF
		
	IF  R6.WaitSecondTick=60  THEN
		//Update the Minute Tick
		R6.WaitMinuteTick:=R6.WaitMinuteTick+1;
		R6.WaitSecondTick:=0;
	END_IF	

	//Update the Remaining Time
	remainingTimeCalculator(elapsedSeconds:= R6.WaitSecondTick, elapsedMinutes:= R6.WaitMinuteTick, givenDuration:= DINT_TO_INT(R6.RecipeStep[R6.R6STEPS].WaitDuration), 
							leftOverSeconds=> R6.RecipeStep[R6.R6STEPS].WaitRemainingSeconds, leftOverMinutes=> R6.RecipeStep[R6.R6STEPS].WaitRemainingMinutes);
	R6.RecipeStep[R6.R6STEPS].WaitRemainingTime := INT_TO_STRING(R6.RecipeStep[R6.R6STEPS].WaitRemainingMinutes);
	R6.RecipeStep[R6.R6STEPS].WaitRemainingTime := CONCAT(STR1:= R6.RecipeStep[R6.R6STEPS].WaitRemainingTime, STR2:= ':');
	R6.RecipeStep[R6.R6STEPS].WaitRemainingTime := CONCAT(STR1:= R6.RecipeStep[R6.R6STEPS].WaitRemainingTime, STR2:= INT_TO_STRING(R6.RecipeStep[R6.R6STEPS].WaitRemainingSeconds));
	
	(*///To write ended time*)
	IF ABS(R6.WaitMinuteTick -R6.RecipeStep[R6.R6STEPS].WaitDuration)=0 THEN
		R6.RecipeStep[R6.R6STEPS].WaitEnded:=TRUE;
		IF R6.RecipeStep[R6.R6STEPS].WaitEndedTime = '' THEN
			R6.RecipeStep[R6.R6STEPS].WaitEndedTime := Main.concatenatedHourMinuteString;
		END_IF
		R6.WaitTick:=0;
		R6.WaitSecondTick:=0;
		R6.WaitMinuteTick:=0;
	END_IF
END_IF
	
IF R6.RecipeStep[R6STEPS].DosingEnabled AND NOT R6.RecipeStep[R6STEPS].DosingEnded THEN
	R6.RecipeStep[R6STEPS].DosingStarted := TRUE;
	IF R6.RecipeStep[R6.R6STEPS].DosingStartedTime = '' THEN
		R6.RecipeStep[R6.R6STEPS].DosingStartedTime := Main.concatenatedHourMinuteString;
	END_IF
	//Update Totalized Volume
		IF  R6.DosingPumpStatus_1 THEN
			DosingTick:=DosingTick+1;
		END_IF
		   
	  IF DosingTick=100 THEN
		  DosingTotalizerVolume:=DosingTotalizerVolume+(R6.RecipeStep[R6STEPS].DosingRateSetpointExpression/2.7 * 0.045);	  
	  END_IF
	  
	  IF DosingTick>100 THEN
		  DosingTick:=0;
	  END_IF
	  
	IF DosingTotalizerVolume < R6.RecipeStep[R6STEPS].DosingMaxAmount THEN
		IF R6.DosingPumpStatus_1 THEN
			IF R6.TemperatureControl < R6.RecipeStep[R6STEPS].DosingStopTemp THEN
				R6.DosingPumpStatus_1 := TRUE;
				R6.DosingPumpSetPoint_1 := R6.RecipeStep[R6STEPS].DosingRateSetpointExpression;
			ELSE
				R6.DosingPumpStatus_1 := FALSE;
				R6.DosingPumpSetPoint_1 := 0;
			END_IF
		ELSE
			IF DosingTotalizerVolume = 0 AND R6.TemperatureControl > R6.RecipeStep[R6STEPS].DosingResumeTemp AND R6.TemperatureControl < R6.RecipeStep[R6STEPS].DosingStopTemp THEN
				//Logic for starting Dosing Pump First Time in a Recipe Step
				R6.DosingPumpStatus_1 := TRUE;
				R6.DosingPumpSetPoint_1 := R6.RecipeStep[R6STEPS].DosingRateSetpointExpression;
			END_IF
			
			IF R6.TemperatureControl < R6.RecipeStep[R6STEPS].DosingResumeTemp THEN
				R6.DosingPumpStatus_1 := TRUE;
				R6.DosingPumpSetPoint_1 := R6.RecipeStep[R6STEPS].DosingRateSetpointExpression;
			END_IF
		END_IF
	ELSE
		R6.DosingPumpStatus_1 := FALSE;
		R6.DosingPumpSetPoint_1 := 0;
		R6.RecipeStep[R6STEPS].DosingEnded := TRUE;
		IF R6.RecipeStep[R6.R6STEPS].DosingEndedTime = '' THEN
			R6.RecipeStep[R6.R6STEPS].DosingEndedTime := Main.concatenatedHourMinuteString;
		END_IF
		DosingTick := 0;
		DosingTotalizerVolume:=0;
	END_IF
END_IF

IF R6.R6STEPS>0 THEN 

(*//Step control block To increment to next step*)
 R6.TotalEnabledValue:=BOOL_TO_INT(R6.RecipeStep[R6.R6STEPS].HeatcoolEnabled)+BOOL_TO_INT(R6.RecipeStep[R6.R6STEPS].StirrerEnabled)+BOOL_TO_INT(R6.RecipeStep[R6.R6STEPS].WaitEnabled)+BOOL_TO_INT( R6.RecipeStep[R6.R6STEPS].DosingEnabled);
 R6.TotalEndedValue:=BOOL_TO_INT(R6.RecipeStep[R6.R6STEPS].HeatCoolEnded)+BOOL_TO_INT(R6.RecipeStep[R6.R6STEPS].StirrerEnded)+BOOL_TO_INT(R6.RecipeStep[R6.R6STEPS].WaitEnded)+BOOL_TO_INT( R6.RecipeStep[R6.R6STEPS].DosingEnded);

    IF (R6.TotalEnabledValue - R6.TotalEndedValue)=0 THEN 
		R6.R6STEPS:=R6.R6STEPS+1;
    END_IF
END_IF
  
 (* ///To End the Recipe**)
 IF  R6.NumberOfRecipeSteps = R6.R6STEPS THEN
	 R6.StirrerStatus:=FALSE;
	 R6.StirrerSetPoint:=0;
	 R6.HeatCoolStatus:=FALSE;
	 R6.HeatCoolSetPoint:=0;	
     R6.StepCompleted:=FALSE;	 
	 R6.RecipeEnded:=TRUE;
	 R6.RecipeStatus:=FALSE;
 END_IF
  
(* //TO ABORT RECIPE*)
AbortTrig(CLK:=R6.AbortRecipe,Q=>);
IF AbortTrig.Q THEN
	shutDownFB(GvlIdentifier := 'R6');
	AbortTrig.CLK := FALSE;
END_IF

END_PROGRAM
